            IF JerkFacLocal <= 0.0 THEN
                JerkFacLocal := 0.1;
            END_IF;

            IF TorqueFacLocal <= 0.0 THEN
                TorqueFacLocal := 0.1;
            END_IF;


            //------------------------------------------------
            // Mapping blending
            //------------------------------------------------
            IF (Item.BlendMode = 0)
               OR (Item.BlendRadius <= 0.0)
            THEN

                BufferMode := C_BM_Buffered;
                TransMode  := C_TM_None;

                TransParam[0] := 0.0;
                TransParam[1] := 0.0;

            ELSE

                //------------------------------------------------
                // Dùng giống MoveP đang chạy ổn
                //------------------------------------------------
                BufferMode := GVL.C_BM_BlendingHigh;

                CASE Item.BlendMode OF

                    1:
                        TransMode := C_TM_CornerDistance;

                    2:
                        TransMode := C_TM_StartVelocity;

                ELSE
                    TransMode := C_TM_CornerDistance;

                END_CASE;

                TransParam[0] := Item.BlendRadius;
                TransParam[1] := 0.0;

            END_IF;


            //------------------------------------------------
            // Orientation mode hiện tại của robot
            //------------------------------------------------
			IF AxisGroup.m_id = SCARA_A.m_id THEN
				OrientationMode := POU_MOTION.RBA_OrientationMode;
			ELSE
				OrientationMode := POU_MOTION.RBB_OrientationMode;
			END_IF
            


            //------------------------------------------------
            // Reset outputs cho command mới
            //------------------------------------------------
            Accepted := FALSE;
            Done     := FALSE;
            Error    := FALSE;
            Timeout  := FALSE;
            Aborted  := FALSE;

            ErrorID_Custom := 0;


            State := E_MoveState.MOVE_SEND;

        END_IF;


    //========================================================
    // SEND COMMAND
    //========================================================
    E_MoveState.MOVE_SEND:

        ExecutePulse := TRUE;

        tAcceptTimeout(
            IN := TRUE,
            PT := AcceptTimeoutTime
        );

        State := E_MoveState.MOVE_WAIT_ACCEPT;


    //========================================================
    // WAIT COMMAND ACCEPTED
    //========================================================
    E_MoveState.MOVE_WAIT_ACCEPT:

        //----------------------------------------------------
        // Giữ Execute cho tới khi AxisGroup nhận command
        //----------------------------------------------------
        ExecutePulse := TRUE;

        tAcceptTimeout(
            IN := TRUE,
            PT := AcceptTimeoutTime
        );


        IF fbMoveL.CommandAccepted THEN

            Accepted := TRUE;

            ExecutePulse := FALSE;

            tAcceptTimeout(IN := FALSE);

            tMoveTimeout(
                IN := TRUE,
                PT := MoveTimeoutTime
            );

            State := E_MoveState.MOVE_WAIT_DONE;


        ELSIF fbMoveL.CommandAborted THEN

            ExecutePulse := FALSE;

            Aborted := TRUE;
            Error   := TRUE;

            ErrorID_Custom := 5103;

            tAcceptTimeout(IN := FALSE);

            State := E_MoveState.MOVE_ABORTED;


        ELSIF fbMoveL.Error THEN

            ExecutePulse := FALSE;

            Error   := TRUE;
            ErrorID := fbMoveL.ErrorID;

            ErrorID_Custom := 5104;

            tAcceptTimeout(IN := FALSE);

            State := E_MoveState.MOVE_ERROR;


        ELSIF tAcceptTimeout.Q THEN

            ExecutePulse := FALSE;

            Timeout := TRUE;
            Error   := TRUE;

            ErrorID_Custom := 5105;

            tAcceptTimeout(IN := FALSE);

            State := E_MoveState.MOVE_TIMEOUT;

        END_IF;


    //========================================================
    // WAIT MOTION DONE
    //========================================================
    E_MoveState.MOVE_WAIT_DONE:

        Accepted := TRUE;
        ExecutePulse := FALSE;

        tMoveTimeout(
            IN := TRUE,
            PT := MoveTimeoutTime
        );


        IF fbMoveL.Done THEN

            tMoveTimeout(IN := FALSE);

            //------------------------------------------------
            // Điểm cần check chính xác
            //------------------------------------------------
            IF NOT Item.SkipPositionCheck THEN

                tPosCheckDelay(
                    IN := TRUE,
                    PT := PosCheckDelayTime
                );

                State := E_MoveState.MOVE_CHECK_POS;

            ELSE

                //------------------------------------------------
                // Điểm transition / blending:
                // không bắt Actual Position == Target.
                //------------------------------------------------
                State := E_MoveState.MOVE_DONE;

            END_IF;


        ELSIF fbMoveL.CommandAborted THEN

            Aborted := TRUE;
            Error   := TRUE;

            ErrorID_Custom := 5103;

            tMoveTimeout(IN := FALSE);

            State := E_MoveState.MOVE_ABORTED;


        ELSIF fbMoveL.Error THEN

            Error   := TRUE;
            ErrorID := fbMoveL.ErrorID;

            ErrorID_Custom := 5104;

            tMoveTimeout(IN := FALSE);

            State := E_MoveState.MOVE_ERROR;


        ELSIF tMoveTimeout.Q THEN

            Timeout := TRUE;
            Error   := TRUE;

            ErrorID_Custom := 5106;

            tMoveTimeout(IN := FALSE);

            State := E_MoveState.MOVE_TIMEOUT;

        END_IF;


    //========================================================
    // CHECK FINAL POSITION
    //========================================================
    E_MoveState.MOVE_CHECK_POS:

        Accepted := TRUE;

        tPosCheckDelay(
            IN := TRUE,
            PT := PosCheckDelayTime
        );

        IF tPosCheckDelay.Q THEN

            tPosCheckDelay(IN := FALSE);

            //------------------------------------------------
            // Lưu để debug
            //------------------------------------------------
// 			IF AxisGroup.m_id = SCARA_A.m_id THEN
//             	DonePosition := POU_MONITOR_ROBOT.RB1_POS;
// 			ELSE
// 				DonePosition := POU_MONITOR_ROBOT.RB2_POS;
// 			END_IF;
			IF AxisGroup.m_id = SCARA_A.m_id THEN
            	DonePosition := POU_COORDINATE_.Pos_Out_A_MCS;
			ELSE
				DonePosition := POU_COORDINATE_.Pos_Out_B_MCS;
			END_IF;


            //------------------------------------------------
            // Kiểm tra vị trí cuối MovL
            //------------------------------------------------
            IF F_CheckPositionReached(
                Target := PosBuf,
                //Actual := POU_MONITOR_ROBOT.RB1_POS,
				Actual := DonePosition,
                TolXYZ := GVL.MotionTolXYZ,
                TolR   := GVL.MotionTolR
            )
            THEN

                State := E_MoveState.MOVE_DONE;

            ELSE

                Error := TRUE;

                //------------------------------------------------
                // 5101 = MoveL position not reached
                //------------------------------------------------
                ErrorID_Custom := 5101;

                State := E_MoveState.MOVE_ERROR;

            END_IF;

        END_IF;


    //========================================================
    // DONE
    //========================================================
    E_MoveState.MOVE_DONE:

        Accepted := TRUE;
        Done     := TRUE;

        ExecutePulse := FALSE;

        //----------------------------------------------------
        // Giống FB_RunMoveP đang dùng:
        // giữ Done cho tới khi Manager đã hạ Start
        // và FB gốc đã hoàn toàn rảnh.
        //----------------------------------------------------
        IF NOT Start
           AND NOT fbMoveL.Busy
           AND NOT fbMoveL.Active
        THEN

            State := E_MoveState.MOVE_IDLE;

        END_IF;


    //========================================================
    // ERROR
    //========================================================
    E_MoveState.MOVE_ERROR:

        Error := TRUE;
        ExecutePulse := FALSE;

        IF NOT Start THEN
            State := E_MoveState.MOVE_IDLE;
        END_IF;


    //========================================================
    // TIMEOUT
    //========================================================
    E_MoveState.MOVE_TIMEOUT:

        Error   := TRUE;
        Timeout := TRUE;

        ExecutePulse := FALSE;

        IF NOT Start THEN
            State := E_MoveState.MOVE_IDLE;
        END_IF;


    //========================================================
    // ABORTED
    //========================================================
    E_MoveState.MOVE_ABORTED:

        Error   := TRUE;
        Aborted := TRUE;

        ExecutePulse := FALSE;

        IF NOT Start THEN
            State := E_MoveState.MOVE_IDLE;
        END_IF;

END_CASE;


//============================================================
// GỌI FB GỐC MỖI SCAN
//============================================================
fbMoveL(
    AxisGroup := AxisGroup,

    Execute := ExecutePulse,

    Position := PosBuf,

    Velocity     := Vel,
    Acceleration := Acc,
    Deceleration := Dec,
    Jerk         := Jerk,

    CoordSystem := CoordSystem,

    BufferMode          := BufferMode,
    TransitionMode      := TransMode,
    TransitionParameter := TransParam,

    OrientationMode := OrientationMode,

    VelFactor    := VelFacLocal,
    AccFactor    := AccFacLocal,
    JerkFactor   := JerkFacLocal,
    TorqueFactor := TorqueFacLocal
);


//============================================================
// PHẢN HỒI TRẠNG THÁI FB GỐC
//============================================================
Busy   := fbMoveL.Busy;
Active := fbMoveL.Active;

END_FUNCTION_BLOCK

// Just_Motion_Control_x86_64_Linux_SM_WV/Application/FB_/FB_RunMoveC
FUNCTION_BLOCK FB_RunMoveC
VAR_INPUT
    Start : BOOL;
    Item  : ST_MotionQueueItem;

    //--------------------------------------------------------
    // Điểm trung gian nằm trên cung
    //--------------------------------------------------------
    MidPosition : SMC_POS_REF;

    //--------------------------------------------------------
    // Điểm cuối cung
    //--------------------------------------------------------
    EndPosition : SMC_POS_REF;

    CoordSystem : SMC_COORD_SYSTEM;

    AcceptTimeoutTime : TIME := T#2S;
    MoveTimeoutTime   : TIME := T#100S;
    PosCheckDelayTime : TIME := T#13MS;
END_VAR

VAR_IN_OUT
    AxisGroup : AXIS_GROUP_REF_SM3;
    //Release   : BOOL;
END_VAR

VAR_OUTPUT
    Accepted       : BOOL;
    Done           : BOOL;
    Busy           : BOOL;
    Active         : BOOL;
    Error          : BOOL;
    Timeout        : BOOL;
    Aborted        : BOOL;

    ErrorID        : SMC_ERROR;
    ErrorID_Custom : INT;

    State          : E_MoveState;
END_VAR

VAR
    //--------------------------------------------------------
    // SoftMotion FB
    //--------------------------------------------------------
    fbMoveC : MC_MoveCircularAbsolute;

    //--------------------------------------------------------
    // Timer
    //--------------------------------------------------------
    tAcceptTimeout : TON;
    tMoveTimeout   : TON;
    tPosCheckDelay : TON;

    //--------------------------------------------------------
    // Execute
    //--------------------------------------------------------
    StartEdge    : BOOL;
    LastStart    : BOOL;
    ExecutePulse : BOOL;

    //--------------------------------------------------------
    // Position buffer
    //--------------------------------------------------------
    MidBuf       : SMC_POS_REF;
    EndBuf       : SMC_POS_REF;
    DonePosition : SMC_POS_REF;

    //--------------------------------------------------------
    // Path dynamics
    //--------------------------------------------------------
    Vel  : LREAL;
    Acc  : LREAL;
    Dec  : LREAL;
    Jerk : LREAL;

    //--------------------------------------------------------
    // Circular parameters
    //--------------------------------------------------------
    CircModeLocal :
        SM3_Robotics.SMC_CIRC_MODE;

    PathChoiceLocal :
        SM3_Robotics.MC_CIRC_PATHCHOICE;

    //--------------------------------------------------------
    // Blending
    //--------------------------------------------------------
    BufferMode :
        SM3_Robotics.MC_BUFFER_MODE;

    TransMode :
        SM3_Robotics.MC_TRANSITION_MODE;

    TransParam :
        ARRAY[0..(SMC_RCNST.MAX_TRANS_PARAMS - 1)] OF LREAL
        := [0.0, 0.0];

    //--------------------------------------------------------
    // Orientation
    //--------------------------------------------------------
    OrientationMode :
        SM3_Robotics.SMC_ORIENTATION_MODE;

    //--------------------------------------------------------
    // Factor
    //--------------------------------------------------------
    VelFacLocal    : LREAL;
    AccFacLocal    : LREAL;
    JerkFacLocal   : LREAL;
    TorqueFacLocal : LREAL;
END_VAR

VAR CONSTANT
    C_BM_Buffered :
        SM3_Robotics.MC_BUFFER_MODE := 1;

    C_TM_CornerDistance :
        SM3_Robotics.MC_TRANSITION_MODE := 2;

    C_TM_None :
        SM3_Robotics.MC_TRANSITION_MODE := 0;

    C_TM_StartVelocity :
        SM3_Robotics.MC_TRANSITION_MODE := 1;
END_VAR

//============================================================
// FB_RunMoveC
//
// Quỹ đạo:
// Current Position → MidPosition → EndPosition
//
// CircMode = BORDER:
// MidPosition là điểm nằm trên cung.
//
// Cơ chế Accepted / Done / Error giống FB_RunMoveP.
//============================================================


//------------------------------------------------------------
// Start edge
//------------------------------------------------------------
StartEdge := Start AND NOT LastStart;
LastStart := Start;


//------------------------------------------------------------
// Execute mặc định FALSE
//------------------------------------------------------------
ExecutePulse := FALSE;


//============================================================
// STATE MACHINE
//============================================================
CASE State OF


    //========================================================
    // IDLE
    //========================================================
    E_MoveState.MOVE_IDLE:

        Accepted := FALSE;
        Done     := FALSE;
        Error    := FALSE;
        Timeout  := FALSE;
        Aborted  := FALSE;

        //Release := FALSE;

        ErrorID_Custom := 0;

        //----------------------------------------------------
        // Reset timer
        //----------------------------------------------------
        tAcceptTimeout(IN := FALSE);
        tMoveTimeout(IN := FALSE);
        tPosCheckDelay(IN := FALSE);


        //----------------------------------------------------
        // Chỉ nhận command khi FB rảnh
        //----------------------------------------------------
        IF Start
           AND NOT fbMoveC.Busy
           AND NOT fbMoveC.Active
        THEN

            //------------------------------------------------
            // Chốt điểm giữa và điểm cuối
            //------------------------------------------------
            MidBuf := MidPosition;
            EndBuf := EndPosition;


            //------------------------------------------------
            // Dynamics
            //------------------------------------------------
           	
			IF Item.Speed > 0.0 THEN
                Vel := Item.Speed;
            ELSE
				IF AxisGroup.m_id = SCARA_A.m_id THEN
                	Vel := GVL.A_CurrentMotionParam.Speed;
				ELSE
					Vel := GVL.B_CurrentMotionParam.Speed;
				END_IF
            END_IF;

            IF AxisGroup.m_id = SCARA_A.m_id THEN
				IF Item.Acceleration > 0.0 THEN Acc := Item.Acceleration; ELSE Acc := GVL_1.DATA_RB_A.MOTION_ACC; END_IF;
				IF Item.Deceleration > 0.0 THEN Dec := Item.Deceleration; ELSE Dec := GVL_1.DATA_RB_A.MOTION_DEC; END_IF;
				IF Item.Jerk > 0.0 THEN Jerk := Item.Jerk; ELSE Jerk := GVL_1.DATA_RB_A.MOTION_JERK; END_IF;
			ELSE
				IF Item.Acceleration > 0.0 THEN Acc := Item.Acceleration; ELSE Acc := GVL_1.DATA_RB_B.MOTION_ACC; END_IF;
				IF Item.Deceleration > 0.0 THEN Dec := Item.Deceleration; ELSE Dec := GVL_1.DATA_RB_B.MOTION_DEC; END_IF;
				IF Item.Jerk > 0.0 THEN Jerk := Item.Jerk; ELSE Jerk := GVL_1.DATA_RB_B.MOTION_JERK; END_IF;
			END_IF


            //------------------------------------------------
            // Fallback
            //------------------------------------------------
            IF Vel <= 0.0 THEN
                Vel := 100.0;
            END_IF;

            IF Acc <= 0.0 THEN
                Acc := 1000.0;
            END_IF;

            IF Dec <= 0.0 THEN
                Dec := 1000.0;
            END_IF;

            IF Jerk <= 0.0 THEN
                Jerk := 10000.0;
            END_IF;


            //------------------------------------------------
            // Factor
            //------------------------------------------------
            IF AxisGroup.m_id = SCARA_A.m_id THEN
				VelFacLocal    := GVL_1.DATA_RB_A.Fac_Vel;
				AccFacLocal    := GVL_1.DATA_RB_A.Fac_Acc;
				JerkFacLocal   := GVL_1.DATA_RB_A.Fac_Jerk;
				TorqueFacLocal := GVL_1.DATA_RB_A.Fac_Torque;
			ELSE
				VelFacLocal    := GVL_1.DATA_RB_B.Fac_Vel;
				AccFacLocal    := GVL_1.DATA_RB_B.Fac_Acc;
				JerkFacLocal   := GVL_1.DATA_RB_B.Fac_Jerk;
				TorqueFacLocal := GVL_1.DATA_RB_B.Fac_Torque;
			END_IF

            IF VelFacLocal <= 0.0 THEN
                VelFacLocal := 0.1;
            END_IF;

            IF AccFacLocal <= 0.0 THEN
                AccFacLocal := 0.1;
            END_IF;

            IF JerkFacLocal <= 0.0 THEN
                JerkFacLocal := 0.1;
            END_IF;

            IF TorqueFacLocal <= 0.0 THEN
                TorqueFacLocal := 0.1;
            END_IF;


            //------------------------------------------------
            // CIRCULAR MODE
            //
            // MidPosition được dạy như điểm nằm trên cung.
            //------------------------------------------------
            CircModeLocal :=
                SM3_Robotics.SMC_CIRC_MODE.BORDER;

            //------------------------------------------------
            // BORDER không dùng PathChoice,
            // nhưng input FB vẫn phải có giá trị hợp lệ.
            //------------------------------------------------
            PathChoiceLocal :=
                SM3_Robotics.MC_CIRC_PATHCHOICE.CLOCKWISE;


            //------------------------------------------------
            // Mapping Blend giống MoveP / MoveL
            //------------------------------------------------
            IF (Item.BlendMode = 0)
               OR (Item.BlendRadius <= 0.0)
            THEN

                BufferMode := C_BM_Buffered;
                TransMode  := C_TM_None;

                TransParam[0] := 0.0;
                TransParam[1] := 0.0;

            ELSE

                BufferMode := GVL.C_BM_BlendingHigh;

                CASE Item.BlendMode OF

                    1:
                        TransMode := C_TM_CornerDistance;

                    2:
                        TransMode := C_TM_StartVelocity;

                ELSE
                    TransMode := C_TM_CornerDistance;

                END_CASE;

                TransParam[0] := Item.BlendRadius;
                TransParam[1] := 0.0;

            END_IF;


            //------------------------------------------------
            // Orientation
            //------------------------------------------------
            IF AxisGroup.m_id = SCARA_A.m_id THEN
				OrientationMode := POU_MOTION.RBA_OrientationMode;
			ELSE
				OrientationMode := POU_MOTION.RBB_OrientationMode;
			END_IF


            //------------------------------------------------
            // Reset outputs
            //------------------------------------------------
            Accepted := FALSE;
            Done     := FALSE;
            Error    := FALSE;
            Timeout  := FALSE;
            Aborted  := FALSE;

            ErrorID_Custom := 0;


            State := E_MoveState.MOVE_SEND;

        END_IF;


    //========================================================
    // SEND COMMAND
    //========================================================
    E_MoveState.MOVE_SEND:

        ExecutePulse := TRUE;

        tAcceptTimeout(
            IN := TRUE,
            PT := AcceptTimeoutTime
        );

        State := E_MoveState.MOVE_WAIT_ACCEPT;


    //========================================================
    // WAIT ACCEPT
    //========================================================
    E_MoveState.MOVE_WAIT_ACCEPT:

        ExecutePulse := TRUE;

        tAcceptTimeout(
            IN := TRUE,
            PT := AcceptTimeoutTime
        );


        IF fbMoveC.CommandAccepted THEN

            Accepted := TRUE;

            ExecutePulse := FALSE;

            tAcceptTimeout(IN := FALSE);

            tMoveTimeout(
                IN := TRUE,
                PT := MoveTimeoutTime
            );

            State := E_MoveState.MOVE_WAIT_DONE;


        ELSIF fbMoveC.CommandAborted THEN

            ExecutePulse := FALSE;

            Aborted := TRUE;
            Error   := TRUE;

            ErrorID_Custom := 5203;

            tAcceptTimeout(IN := FALSE);

            State := E_MoveState.MOVE_ABORTED;


        ELSIF fbMoveC.Error THEN

            ExecutePulse := FALSE;

            Error   := TRUE;
            ErrorID := fbMoveC.ErrorID;

            ErrorID_Custom := 5204;

            tAcceptTimeout(IN := FALSE);

            State := E_MoveState.MOVE_ERROR;


        ELSIF tAcceptTimeout.Q THEN

            ExecutePulse := FALSE;

            Timeout := TRUE;
            Error   := TRUE;

            ErrorID_Custom := 5205;

            tAcceptTimeout(IN := FALSE);

            State := E_MoveState.MOVE_TIMEOUT;

        END_IF;


    //========================================================
    // WAIT DONE
    //========================================================
    E_MoveState.MOVE_WAIT_DONE:

        Accepted := TRUE;
        ExecutePulse := FALSE;

        tMoveTimeout(
            IN := TRUE,
            PT := MoveTimeoutTime
        );


        IF fbMoveC.Done THEN

            tMoveTimeout(IN := FALSE);

            //------------------------------------------------
            // MovC chỉ check vị trí cuối EndBuf.
            //
            // MidBuf tuyệt đối không check vì đó chỉ là điểm
            // dùng để xác định hình học của cung.
            //------------------------------------------------
            IF NOT Item.SkipPositionCheck THEN

                tPosCheckDelay(
                    IN := TRUE,
                    PT := PosCheckDelayTime
                );

                State := E_MoveState.MOVE_CHECK_POS;

            ELSE

                State := E_MoveState.MOVE_DONE;

            END_IF;


        ELSIF fbMoveC.CommandAborted THEN

            Aborted := TRUE;
            Error   := TRUE;

            ErrorID_Custom := 5203;

            tMoveTimeout(IN := FALSE);

            State := E_MoveState.MOVE_ABORTED;


        ELSIF fbMoveC.Error THEN

            Error   := TRUE;
            ErrorID := fbMoveC.ErrorID;

            ErrorID_Custom := 5204;

            tMoveTimeout(IN := FALSE);

            State := E_MoveState.MOVE_ERROR;


        ELSIF tMoveTimeout.Q THEN

            Timeout := TRUE;
            Error   := TRUE;

            ErrorID_Custom := 5206;

            tMoveTimeout(IN := FALSE);

            State := E_MoveState.MOVE_TIMEOUT;

        END_IF;


    //========================================================
    // CHECK END POSITION
    //========================================================
    E_MoveState.MOVE_CHECK_POS:

        Accepted := TRUE;

        tPosCheckDelay(
            IN := TRUE,
            PT := PosCheckDelayTime
        );

        IF tPosCheckDelay.Q THEN

            tPosCheckDelay(IN := FALSE);

            //------------------------------------------------
            // Lưu để debug
            //------------------------------------------------
//             IF AxisGroup.m_id = SCARA_A.m_id THEN
//             	DonePosition := POU_MONITOR_ROBOT.RB1_POS;
// 			ELSE
// 				DonePosition := POU_MONITOR_ROBOT.RB2_POS;
// 			END_IF;
			
			IF AxisGroup.m_id = SCARA_A.m_id THEN
            	DonePosition := POU_COORDINATE_.Pos_Out_A_MCS;
			ELSE
				DonePosition := POU_COORDINATE_.Pos_Out_B_MCS;
			END_IF;



            //------------------------------------------------
            // Với MoveC chỉ kiểm tra END POINT.
            //------------------------------------------------
            IF F_CheckPositionReached(
                Target := EndBuf,
                //Actual := POU_MONITOR_ROBOT.RB1_POS,
				Actual := DonePosition,
                TolXYZ := GVL.MotionTolXYZ,
                TolR   := GVL.MotionTolR
            )
            THEN

                State := E_MoveState.MOVE_DONE;

            ELSE

                Error := TRUE;

                //------------------------------------------------
                // 5201 = Circular end position not reached
                //------------------------------------------------
                ErrorID_Custom := 5201;

                State := E_MoveState.MOVE_ERROR;

            END_IF;

        END_IF;


    //========================================================
    // DONE
    //========================================================
    E_MoveState.MOVE_DONE:

        Accepted := TRUE;
        Done     := TRUE;

        ExecutePulse := FALSE;

        IF NOT Start
           AND NOT fbMoveC.Busy
           AND NOT fbMoveC.Active
        THEN

            State := E_MoveState.MOVE_IDLE;

        END_IF;


    //========================================================
    // ERROR
    //========================================================
    E_MoveState.MOVE_ERROR:

        Error := TRUE;
        ExecutePulse := FALSE;

        IF NOT Start THEN
            State := E_MoveState.MOVE_IDLE;
        END_IF;


    //========================================================
    // TIMEOUT
    //========================================================
    E_MoveState.MOVE_TIMEOUT:

        Error   := TRUE;
        Timeout := TRUE;

        ExecutePulse := FALSE;

        IF NOT Start THEN
            State := E_MoveState.MOVE_IDLE;
        END_IF;


    //========================================================
    // ABORTED
    //========================================================
    E_MoveState.MOVE_ABORTED:

        Error   := TRUE;
        Aborted := TRUE;

        ExecutePulse := FALSE;

        IF NOT Start THEN
            State := E_MoveState.MOVE_IDLE;
        END_IF;

END_CASE;


//============================================================
// GỌI FB GỐC MỖI SCAN
//============================================================
fbMoveC(
    AxisGroup := AxisGroup,

    Execute := ExecutePulse,

    //--------------------------------------------------------
    // Dùng BORDER:
    // MidBuf là điểm nằm trên cung.
    //--------------------------------------------------------
    CircMode := CircModeLocal,
    AuxPoint := MidBuf,
    EndPoint := EndBuf,

    PathChoice := PathChoiceLocal,

    Velocity     := Vel,
    Acceleration := Acc,
    Deceleration := Dec,
    Jerk         := Jerk,

    CoordSystem := CoordSystem,

    BufferMode          := BufferMode,
    TransitionMode      := TransMode,
    TransitionParameter := TransParam,

    OrientationMode := OrientationMode,

    VelFactor    := VelFacLocal,
    AccFactor    := AccFacLocal,
    JerkFactor   := JerkFacLocal,
    TorqueFactor := TorqueFacLocal
);


//============================================================
// PHẢN HỒI FB GỐC
//============================================================
Busy   := fbMoveC.Busy;
Active := fbMoveC.Active;

END_FUNCTION_BLOCK

// Just_Motion_Control_x86_64_Linux_SM_WV/Application/FB_/Vision/FB_VisionAlign
FUNCTION_BLOCK FB_VisionAlign
VAR_INPUT
    Enable : BOOL;                              // Cho phép FB hoạt động.
    Start : BOOL;                               // Bắt đầu một lần Align.
    CameraID : UINT;                            // Camera sử dụng.
    JobID : UINT;                               // Job Vision Align.
END_VAR

VAR_OUTPUT
    Busy : BOOL;                                // Đang chạy.
    Done : BOOL;                                // Hoàn thành.
    Error : BOOL;                               // Có lỗi.
    ErrorID : INT;                              // Mã lỗi.
    State : INT;                                // State monitor.

    HeaderOK : BOOL;                            // Đã nhận Header hợp lệ.
    TriggerID : UDINT;                          // TriggerID của Result.

    VisionX : REAL;                             // X Vision trả về.
    VisionY : REAL;                             // Y Vision trả về.
    VisionZ : REAL;                             // Z Vision trả về.
    VisionA : REAL;                             // Theta Vision trả về.
    VisionScore : REAL;                         // Score Vision.
    VisionFeatureID : UINT;                     // FeatureID Vision.

    ResultValid : BOOL;                         // Valid từ Vision.
    ResultStatus : E_VisionResultStatus;        // Status Vision.
END_VAR

VAR
    StartOld : BOOL;                            // Start scan trước.
    xStartVision : BOOL;                        // Start FB VisionGetResult.

    fbVisionGetResult : FB_VisionGetResult;     // FB Trigger + nhận Result.
END_VAR

//=============================================================================
// FB_VisionAlign - SIMPLE VERSION
//-----------------------------------------------------------------------------
// FB này không tự xử lý Modbus.
// Không tự gọi FB_TriggerVS / FB_VisionWaitResult.
// Toàn bộ Trigger + nhận Result giao cho FB_VisionGetResult.
//=============================================================================


//=============================================================================
// CALL FB VISION GET RESULT
//=============================================================================
fbVisionGetResult(
    Enable := Enable,
    Start := xStartVision,
    CameraID := CameraID,
    JobID := JobID,
    Application := E_VisionApplication.VIS_APP_ALIGN
);


//=============================================================================
// RESET
//=============================================================================
IF NOT Enable THEN
    State := 0;
    StartOld := FALSE;
    xStartVision := FALSE;

    Busy := FALSE;
    Done := FALSE;
    Error := FALSE;
    ErrorID := 0;

    HeaderOK := FALSE;
    TriggerID := 0;

    VisionX := 0.0;
    VisionY := 0.0;
    VisionZ := 0.0;
    VisionA := 0.0;
    VisionScore := 0.0;
    VisionFeatureID := 0;

    ResultValid := FALSE;
    ResultStatus := E_VisionResultStatus.VIS_RESULT_NONE;

    RETURN;
END_IF;


//=============================================================================
// STATE MACHINE
//=============================================================================
CASE State OF

    //=========================================================================
    // 0 - IDLE
    //=========================================================================
    0:
        Busy := FALSE;
        Done := FALSE;
        Error := FALSE;
        ErrorID := 0;

        xStartVision := FALSE;
        HeaderOK := FALSE;

        IF Start AND NOT StartOld THEN
            Busy := TRUE;

            xStartVision := TRUE;

            State := 10;
        END_IF;


    //=========================================================================
    // 10 - WAIT VISION RESULT
    //=========================================================================
    10:
        Busy := TRUE;

        IF fbVisionGetResult.Error THEN
            xStartVision := FALSE;

            Error := TRUE;
            ErrorID := fbVisionGetResult.ErrorID;

            State := 900;

        ELSIF fbVisionGetResult.Done THEN
            xStartVision := FALSE;

            State := 20;
        END_IF;


    //=========================================================================
    // 20 - COPY VISION RESULT
    //=========================================================================
    20:
        HeaderOK := fbVisionGetResult.HeaderOK;
        TriggerID := fbVisionGetResult.TriggerID;

        VisionX := fbVisionGetResult.X;
        VisionY := fbVisionGetResult.Y;
        VisionZ := fbVisionGetResult.Z;
        VisionA := fbVisionGetResult.A;
        VisionScore := fbVisionGetResult.Score;
        VisionFeatureID := fbVisionGetResult.FeatureID;

        ResultValid := fbVisionGetResult.ResultValid;
        ResultStatus := fbVisionGetResult.ResultStatus;

        State := 30;


    //=========================================================================
    // 30 - ALIGN RESULT READY
    //-------------------------------------------------------------------------
    // Hiện tại chưa xử lý Transform / Correction.
    // Chỉ xác nhận đã nhận được dữ liệu Vision.
    //=========================================================================
    30:
        IF HeaderOK THEN
            Busy := FALSE;
            Done := TRUE;

            State := 100;
        ELSE
            Error := TRUE;
            ErrorID := 301;                  // Không có Header hợp lệ.

            State := 900;
        END_IF;


    //=========================================================================
    // 100 - DONE
    //=========================================================================
    100:
        Busy := FALSE;
        Done := TRUE;

        IF NOT Start THEN
            State := 0;
        END_IF;


    //=========================================================================
    // 900 - ERROR
    //=========================================================================
    900:
        Busy := FALSE;
        Done := FALSE;

        xStartVision := FALSE;

        IF NOT Start THEN
            Error := FALSE;
            ErrorID := 0;

            State := 0;
        END_IF;

END_CASE;


//=============================================================================
// SAVE START
//=============================================================================
StartOld := Start;

END_FUNCTION_BLOCK

// Just_Motion_Control_x86_64_Linux_SM_WV/Application/FB_/Vision/FB_VisionGetResult
FUNCTION_BLOCK FB_VisionGetResult
VAR_INPUT
    Enable : BOOL;                              // Cho phép FB hoạt động.
    Start : BOOL;                               // Cạnh lên bắt đầu một lần đọc Vision.
    CameraID : UINT;                            // Camera sử dụng.
    JobID : UINT;                               // JobID Vision.
    Application : E_VisionApplication;          // Application Vision.
END_VAR

VAR_OUTPUT
    Busy : BOOL;                                // Đang thực hiện.
    Done : BOOL;                                // Đã nhận Result thành công.
    Error : BOOL;                               // Có lỗi.
    ErrorID : INT;                              // Mã lỗi.

    State : INT;                                // State để monitor.

    TriggerID : UDINT;                          // TriggerID của lần chụp.

    HeaderOK : BOOL;                            // TRUE khi Header Result hợp lệ.

    ResultValid : BOOL;                         // Bit Valid của dữ liệu Vision.
    ResultStatus : E_VisionResultStatus;        // ResultStatus Vision.
    ResultCode : UINT;                          // ResultCode Vision.
    VisionErrorCode : UINT;                     // ErrorCode Vision.

    X : REAL;                                   // X Vision trả về.
    Y : REAL;                                   // Y Vision trả về.
    Z : REAL;                                   // Z Vision trả về.
    A : REAL;                                   // Theta / Angle Vision trả về.
    Score : REAL;                               // Score Vision.
    FeatureID : UINT;                           // FeatureID Vision.
END_VAR

VAR
    StartOld : BOOL;                            // Start scan trước.

    xStartTrigger : BOOL;                       // Start nội bộ cho Trigger.
    xStartWaitResult : BOOL;                    // Start nội bộ cho WaitResult.

    fbTriggerVS : FB_TriggerVS;                 // FB Trigger đã test.
    fbWaitResult : FB_VisionWaitResult;         // FB WaitResult đã test.
END_VAR

//=============================================================================
// FB_VisionGetResult
//-----------------------------------------------------------------------------
// Chức năng đơn giản:
// 1. Trigger Vision.
// 2. Chờ Vision trả Result.
// 3. Khi Header hợp lệ và đúng TriggerID thì copy dữ liệu ra Output.
// 4. Không kiểm tra Offset / Tolerance / Motion.
//=============================================================================


//=============================================================================
// CALL TRIGGER
//=============================================================================
fbTriggerVS(
    Enable := Enable,
    Start := xStartTrigger,
    CameraID := CameraID,
    JobID := JobID,
    Application := Application,
    count_Vs_Align_max := GVL.g_aVisionConfig[CameraID].MaxRetry,
    T_Delay_Trigger_time := TO_INT(GVL.g_aVisionConfig[CameraID].TriggerTimeout),
    Trigger_Again := FALSE,
    Pass_Triger_VS_NG := FALSE,
    Mode_ByPass_VS := FALSE
);

TriggerID := fbTriggerVS.CurrentTriggerID;


//=============================================================================
// CALL WAIT RESULT
//=============================================================================
fbWaitResult(
    Enable := Enable,
    Start := xStartWaitResult,
    CameraID := CameraID,
    ExpectedTriggerID := TriggerID,
    ExpectedJobID := JobID,
    ExpectedApplication := Application
);


//=============================================================================
// DISABLE / RESET
//=============================================================================
IF NOT Enable THEN
    State := 0;
    StartOld := FALSE;

    Busy := FALSE;
    Done := FALSE;
    Error := FALSE;
    ErrorID := 0;

    xStartTrigger := FALSE;
    xStartWaitResult := FALSE;

    HeaderOK := FALSE;

    ResultValid := FALSE;
    ResultStatus := E_VisionResultStatus.VIS_RESULT_NONE;
    ResultCode := 0;
    VisionErrorCode := 0;

    X := 0.0;
    Y := 0.0;
    Z := 0.0;
    A := 0.0;
    Score := 0.0;
    FeatureID := 0;

    RETURN;
END_IF;


//=============================================================================
// STATE MACHINE
//=============================================================================
CASE State OF

    //=========================================================================
    // 0 - IDLE
    //=========================================================================
    0:
        Busy := FALSE;
        Done := FALSE;
        Error := FALSE;
        ErrorID := 0;

        xStartTrigger := FALSE;
        xStartWaitResult := FALSE;

        HeaderOK := FALSE;

        IF Start AND NOT StartOld THEN
            Busy := TRUE;
            xStartTrigger := TRUE;
            State := 10;
        END_IF;


    //=========================================================================
    // 10 - WAIT TRIGGER DONE
    //=========================================================================
    10:
        Busy := TRUE;

        IF fbTriggerVS.Error THEN
            xStartTrigger := FALSE;

            Error := TRUE;
            ErrorID := 100 + fbTriggerVS.ErrorID;
            State := 900;

        ELSIF fbTriggerVS.DoneAll THEN
            xStartTrigger := FALSE;

            xStartWaitResult := TRUE;
            State := 20;
        END_IF;


    //=========================================================================
    // 20 - WAIT RESULT
    //=========================================================================
    20:
        Busy := TRUE;

        IF fbWaitResult.Error THEN
            xStartWaitResult := FALSE;

            Error := TRUE;
            ErrorID := 200 + fbWaitResult.ErrorID;
            State := 900;

        ELSIF fbWaitResult.Done THEN
            xStartWaitResult := FALSE;

            State := 30;
        END_IF;


    //=========================================================================
    // 30 - COPY RESULT
    //=========================================================================
    30:
        // Header đã được FB_WaitResult xác nhận đúng TriggerID / JobID / App.
        HeaderOK := TRUE;

        ResultValid := fbWaitResult.ResultValid;
        ResultStatus := fbWaitResult.ResultStatus;
        ResultCode := fbWaitResult.ResultCode;
        VisionErrorCode := fbWaitResult.VisionErrorCode;

        X := fbWaitResult.ResultX;
        Y := fbWaitResult.ResultY;
        Z := fbWaitResult.ResultZ;
        A := fbWaitResult.ResultA;
        Score := fbWaitResult.ResultScore;
        FeatureID := fbWaitResult.ResultFeatureID;

        Busy := FALSE;
        Done := TRUE;

        State := 100;


    //=========================================================================
    // 100 - DONE
    //=========================================================================
    100:
        Busy := FALSE;
        Done := TRUE;

        IF NOT Start THEN
            State := 0;
        END_IF;


    //=========================================================================
    // 900 - ERROR
    //=========================================================================
    900:
        Busy := FALSE;
        Done := FALSE;

        xStartTrigger := FALSE;
        xStartWaitResult := FALSE;

        IF NOT Start THEN
            Error := FALSE;
            ErrorID := 0;
            State := 0;
        END_IF;

END_CASE;

StartOld := Start;

END_FUNCTION_BLOCK

// Just_Motion_Control_x86_64_Linux_SM_WV/Application/FB_/FB_MotionQueuePush_B
FUNCTION_BLOCK FB_MotionQueuePush_B
VAR_INPUT
	Item : ST_MotionQueueItem;
    Execute : BOOL;
END_VAR
VAR_OUTPUT
	Done : BOOL;
    Error : BOOL;
	Busy  : BOOL;
END_VAR
VAR
	ExecuteOld  : BOOL;
	ExecuteRise : BOOL;
END_VAR

//====================================================
// FB_MotionQueuePush
// Execute = TRUE  -> Push đúng 1 lần
// Done/Error giữ đến khi Execute = FALSE
//====================================================

IF NOT Execute THEN

    Done := FALSE;
    Error := FALSE;
    Busy := FALSE;

ELSE

    IF NOT Busy THEN

        Busy := TRUE;

        IF GVL.B_MotionCount >= 20 THEN

            Error := TRUE;
            Done := FALSE;

        ELSE

            GVL.B_MotionQueue[GVL.B_MotionTail] := Item;

            GVL.B_MotionTail := GVL.B_MotionTail + 1;

            IF GVL.B_MotionTail > 20 THEN
                GVL.B_MotionTail := 1;
            END_IF;

            GVL.B_MotionCount := GVL.B_MotionCount + 1;

            Done := TRUE;
            Error := FALSE;

        END_IF;

    END_IF;

END_IF;

END_FUNCTION_BLOCK

// Just_Motion_Control_x86_64_Linux_SM_WV/Application/FB_/FB_MotionQueuePop_B
FUNCTION_BLOCK FB_MotionQueuePop_B
VAR_INPUT
	Execute : BOOL;
END_VAR
VAR_OUTPUT
	Item  : ST_MotionQueueItem;
    Done  : BOOL;
    Empty : BOOL;
	Busy  : BOOL;
END_VAR
VAR
	ExecuteOld  : BOOL;
	ExecuteRise : BOOL;
END_VAR

IF NOT Execute THEN

    Done := FALSE;
    Empty := FALSE;
    Busy := FALSE;

ELSE

    IF NOT Busy THEN

        Busy := TRUE;

        IF GVL.B_MotionCount <= 0 THEN

            Empty := TRUE;
            Done := FALSE;

        ELSE

            Item := GVL.B_MotionQueue[GVL.B_MotionHead];

            GVL.B_MotionHead := GVL.B_MotionHead + 1; // Tang gia tri len 1 sau khi lay

            IF GVL.B_MotionHead > 20 THEN // Nếu Head vượt quá 20 thì quay lại 1
                GVL.B_MotionHead := 1;
            END_IF;

            GVL.B_MotionCount := GVL.B_MotionCount - 1; // giam so luong phan di trong queue di 1

            Done := TRUE;
            Empty := FALSE;

        END_IF;

    END_IF;

END_IF;

END_FUNCTION_BLOCK

// Just_Motion_Control_x86_64_Linux_SM_WV/Application/FC_/F_IsMotionCmd
FUNCTION F_IsMotionCmd : BOOL // Kiem tra xem phai la motion cmd khong
VAR_INPUT
	Cmd : E_RobotCmd;
END_VAR
VAR
END_VAR

CASE Cmd OF
    E_RobotCmd.CMD_MovP,
    E_RobotCmd.CMD_MovL,
    E_RobotCmd.CMD_MovC:
        F_IsMotionCmd := TRUE;
ELSE
    F_IsMotionCmd := FALSE;
END_CASE

END_FUNCTION

// Just_Motion_Control_x86_64_Linux_SM_WV/Application/FC_/RBA/F_EvalCondition_A
FUNCTION F_EvalCondition_A : BOOL
VAR_INPUT
    CondNo : INT;
END_VAR

VAR
    i : INT;
    rowResult : BOOL;
    finalResult : BOOL;
    firstRow : BOOL;
END_VAR

IF (CondNo < 1) OR (CondNo > 100) THEN
    F_EvalCondition_A := FALSE;
    RETURN;
END_IF;

IF NOT GVL_1.Condition_Cr_A[CondNo].Enable THEN
    F_EvalCondition_A := FALSE;
    RETURN;
END_IF;

firstRow := TRUE;
finalResult := FALSE;

FOR i := 1 TO 10 DO

    IF GVL_1.Condition_Cr_A[CondNo].Row[i].Enable THEN

        rowResult := F_EvalCondRow_A(GVL_1.Condition_Cr_A[CondNo].Row[i]);

        IF firstRow THEN
            finalResult := rowResult;
            firstRow := FALSE;
        ELSE
            CASE GVL_1.Condition_Cr_A[CondNo].Row[i - 1].LinkNext OF
                1: finalResult := finalResult AND rowResult;
                2: finalResult := finalResult OR rowResult;
            ELSE
                finalResult := finalResult AND rowResult;
            END_CASE;
        END_IF;

    END_IF;

END_FOR;

GVL_1.Condition_Cr_A[CondNo].Result := finalResult;
F_EvalCondition_A := finalResult;

END_FUNCTION

// Just_Motion_Control_x86_64_Linux_SM_WV/Application/FC_/RBA/F_EvalCondRow_A
FUNCTION F_EvalCondRow_A : BOOL
VAR_INPUT
    Row : ST_ConditionRow;
END_VAR

VAR
    actualValue : LREAL;
END_VAR

IF NOT Row.Enable THEN
    F_EvalCondRow_A := TRUE;
    RETURN;
END_IF;

actualValue := F_GetCondValue_A(
    Source := Row.Source,
    Index  := Row.Index
);

CASE Row.Operator OF
    1: F_EvalCondRow_A := actualValue = Row.SetValue;
    2: F_EvalCondRow_A := actualValue <> Row.SetValue;
    3: F_EvalCondRow_A := actualValue > Row.SetValue;
    4: F_EvalCondRow_A := actualValue >= Row.SetValue;
    5: F_EvalCondRow_A := actualValue < Row.SetValue;
    6: F_EvalCondRow_A := actualValue <= Row.SetValue;
ELSE
    F_EvalCondRow_A := FALSE;
END_CASE;

END_FUNCTION

// Just_Motion_Control_x86_64_Linux_SM_WV/Application/FC_/RBA/F_GetCondValue_A
FUNCTION F_GetCondValue_A : DINT
VAR_INPUT
    Source : INT;
    Index  : INT;
END_VAR

CASE Source OF
	0:
    1: // DI
        IF GVL.X[Index] THEN
            F_GetCondValue_A := 1;
        ELSE
            F_GetCondValue_A := 0;
        END_IF;

    2: // DO
        IF GVL.Y[Index] THEN
            F_GetCondValue_A := 1;
        ELSE
            F_GetCondValue_A := 0;
        END_IF;

//     3: // REG
//         F_GetCondValue_A := GVL.A_Reg[Index];
// 
//     4: // VAR
//         F_GetCondValue_A := GVL.A_Var[Index];

ELSE
    F_GetCondValue_A := 0;

END_CASE;

END_FUNCTION

// Just_Motion_Control_x86_64_Linux_SM_WV/Application/FC_/RBA/F_FindElseOrEndIf_A
FUNCTION F_FindElseOrEndIf_A : INT
VAR_INPUT
    StartStep : INT;
END_VAR

VAR
    i : INT;
    depth : INT;
    cmd : E_RobotCmd;
END_VAR

//====================================================
// Tìm ELSE hoặc END_IF tương ứng với IF tại StartStep
// Có hỗ trợ IF lồng nhau
//====================================================

depth := 0;

FOR i := StartStep + 1 TO GVL.A_LengthStep DO

    cmd := GVL_1.Step_Cr_A[i].Cmd;

    CASE cmd OF

        E_RobotCmd.CMD_IF,
        E_RobotCmd.CMD_IF_IN,
        E_RobotCmd.CMD_IF_VAR,
        E_RobotCmd.CMD_IF_REG:
            depth := depth + 1;


        E_RobotCmd.CMD_END_IF:
            IF depth = 0 THEN
                // Không có ELSE, nhảy tới sau END_IF
                F_FindElseOrEndIf_A := i + 1;
                RETURN;
            ELSE
                depth := depth - 1;
            END_IF;


        E_RobotCmd.CMD_ELSE:
            IF depth = 0 THEN
                // Có ELSE, nhảy tới step sau ELSE
                F_FindElseOrEndIf_A := i + 1;
                RETURN;
            END_IF;

    END_CASE;

END_FOR;

// Không tìm thấy thì báo về cuối chương trình
F_FindElseOrEndIf_A := GVL.A_LengthStep + 1;

END_FUNCTION

// Just_Motion_Control_x86_64_Linux_SM_WV/Application/FC_/RBA/F_CompareDINT_A
FUNCTION F_CompareDINT_A : BOOL
VAR_INPUT
	Actual   : DINT;
    Operator : DINT;
    SetValue : DINT;
END_VAR
VAR
END_VAR

CASE Operator OF
    1: F_CompareDINT_A := Actual =  SetValue;
    2: F_CompareDINT_A := Actual <> SetValue;
    3: F_CompareDINT_A := Actual >  SetValue;
    4: F_CompareDINT_A := Actual >= SetValue;
    5: F_CompareDINT_A := Actual <  SetValue;
    6: F_CompareDINT_A := Actual <= SetValue;
ELSE
    F_CompareDINT_A := FALSE;
END_CASE;

END_FUNCTION

// Just_Motion_Control_x86_64_Linux_SM_WV/Application/FC_/RBA/F_FindEndIf_A
FUNCTION F_FindEndIf_A : INT
VAR_INPUT
    StartStep : INT;
END_VAR

VAR
    i : INT;
    depth : INT;
    cmd : E_RobotCmd;
END_VAR

//====================================================
// Tìm END_IF tương ứng với ELSE hiện tại
// Có hỗ trợ IF lồng nhau
//====================================================

depth := 0;

FOR i := StartStep + 1 TO GVL.A_LengthStep DO

    cmd := GVL_1.Step_Cr_A[i].Cmd;

    CASE cmd OF

        E_RobotCmd.CMD_IF,
        E_RobotCmd.CMD_IF_IN,
        E_RobotCmd.CMD_IF_VAR,
        E_RobotCmd.CMD_IF_REG:
			// gặp IF con trong nhánh ELSE
            depth := depth + 1;


        E_RobotCmd.CMD_END_IF:
            IF depth = 0 THEN
                // Nhảy tới sau END_IF, END_IF tương ứng với ELSE hiện tại
                F_FindEndIf_A := i + 1;
                RETURN;
            ELSE
                depth := depth - 1;
            END_IF;

    END_CASE;

END_FOR;

F_FindEndIf_A := GVL.A_LengthStep + 1;

END_FUNCTION

// Just_Motion_Control_x86_64_Linux_SM_WV/Application/FC_/RBA/F_FindEndWhile_A
FUNCTION F_FindEndWhile_A : INT
VAR_INPUT
    StartStep : INT;
END_VAR

VAR
    i : INT;
    depth : INT;
    cmd : E_RobotCmd;
END_VAR

//====================================================
// Tìm END_WHILE tương ứng với WHILE tại StartStep
// Có hỗ trợ WHILE lồng nhau
//====================================================

depth := 0;

FOR i := StartStep + 1 TO GVL.A_LengthStep DO

    cmd := GVL_1.Step_Cr_A[i].Cmd;

    CASE cmd OF

        E_RobotCmd.CMD_WHILE,
        E_RobotCmd.CMD_WHILE_IN,
        E_RobotCmd.CMD_WHILE_REG:
            depth := depth + 1;


        E_RobotCmd.CMD_END_WHILE:
            IF depth = 0 THEN
                // WHILE sai, nhảy tới sau END_WHILE
                F_FindEndWhile_A := i + 1;
                RETURN;
            ELSE
                depth := depth - 1;
            END_IF;

    END_CASE;

END_FOR;

F_FindEndWhile_A := GVL.A_LengthStep + 1;

END_FUNCTION

// Just_Motion_Control_x86_64_Linux_SM_WV/Application/FC_/RBA/F_FindWhileStart_A
FUNCTION F_FindWhileStart_A : INT
VAR_INPUT
    EndWhileStep : INT;
END_VAR

VAR
    i : INT;
    depth : INT;
    cmd : E_RobotCmd;
END_VAR

//====================================================
// Tìm WHILE tương ứng khi đang đứng tại END_WHILE
// Quét ngược và hỗ trợ WHILE lồng nhau
//====================================================

depth := 0;

FOR i := EndWhileStep - 1 TO 1 BY -1 DO

    cmd := GVL_1.Step_Cr_A[i].Cmd;

    CASE cmd OF

        E_RobotCmd.CMD_END_WHILE:
            depth := depth + 1;


        E_RobotCmd.CMD_WHILE,
        E_RobotCmd.CMD_WHILE_IN,
        E_RobotCmd.CMD_WHILE_REG:
            IF depth = 0 THEN
                F_FindWhileStart_A := i;
                RETURN;
            ELSE
                depth := depth - 1;
            END_IF;

    END_CASE;

END_FOR;

F_FindWhileStart_A := 1;




// E_RobotCmd.CMD_ELSE:
//     // Nếu đã chạy nhánh IF TRUE, gặp ELSE thì bỏ qua ELSE block
//     GVL.A_RunStep := F_FindEndIf_A(GVL.A_RunStep);
//     GVL.A_RunState := 0;
// 

// E_RobotCmd.CMD_END_IF:
//     // Kết thúc IF block
//     GVL.A_RunStep := GVL.A_RunStep + 1;
//     GVL.A_RunState := 0;
// 
// 
// E_RobotCmd.CMD_WHILE:
//     // P1 = Condition No
//     IF F_EvalCondition_A(step_PRG_A_Interpreter.P1) THEN
//         GVL.A_RunStep := GVL.A_RunStep + 1;
//     ELSE
//         GVL.A_RunStep := F_FindEndWhile_A(GVL.A_RunStep);
//     END_IF;
// 
//     GVL.A_RunState := 0;
// 
// 
// E_RobotCmd.CMD_END_WHILE:
//     // Quay lại đầu WHILE để kiểm tra điều kiện lại
//     GVL.A_RunStep := F_FindWhileStart_A(GVL.A_RunStep);
//     GVL.A_RunState := 0;

END_FUNCTION

// Just_Motion_Control_x86_64_Linux_SM_WV/Application/FC_/RBA/F_CalcReg_A
FUNCTION F_CalcReg_A : DINT
VAR_INPUT
    Cmd       : E_RobotCmd;
    DestReg   : DINT;
    SourceMode: DINT;
    P3        : DINT;
    P4        : DINT;
END_VAR

VAR
    A : DINT;
    B : DINT;
END_VAR

//====================================================
// SourceMode:
// 0: RegDest với số cố định P3
// 1: RegDest với Reg[P3]
// 2: Reg[P3] với Reg[P4], trả về RegDest
//====================================================

IF (DestReg < 1) OR (DestReg > 200) THEN
    F_CalcReg_A := 0;
    RETURN;
END_IF;

CASE SourceMode OF

    0:
        A := GVL.A_Reg[DestReg];
        B := P3;

    1:
        A := GVL.A_Reg[DestReg];

        IF (P3 >= 1) AND (P3 <= 200) THEN
            B := GVL.A_Reg[P3];
        ELSE
            B := 0;
        END_IF;

    2:
        IF (P3 >= 1) AND (P3 <= 200) THEN
            A := GVL.A_Reg[P3];
        ELSE
            A := 0;
        END_IF;

        IF (P4 >= 1) AND (P4 <= 200) THEN
            B := GVL.A_Reg[P4];
        ELSE
            B := 0;
        END_IF;

ELSE
    A := GVL.A_Reg[DestReg];
    B := 0;

END_CASE;


CASE Cmd OF

    E_RobotCmd.CMD_REG_SET:
        F_CalcReg_A := B;

    E_RobotCmd.CMD_REG_ADD:
        F_CalcReg_A := A + B;

    E_RobotCmd.CMD_REG_SUB:
        F_CalcReg_A := A - B;

    E_RobotCmd.CMD_REG_MUL:
        F_CalcReg_A := A * B;

    E_RobotCmd.CMD_REG_DIV:
        IF B <> 0 THEN
            F_CalcReg_A := A / B;
        ELSE
            F_CalcReg_A := GVL.A_Reg[DestReg];
        END_IF;

    E_RobotCmd.CMD_REG_MOD:
        IF B <> 0 THEN
            F_CalcReg_A := A MOD B;
        ELSE
            F_CalcReg_A := GVL.A_Reg[DestReg];
        END_IF;

ELSE
    F_CalcReg_A := GVL.A_Reg[DestReg];

END_CASE;

END_FUNCTION

// Just_Motion_Control_x86_64_Linux_SM_WV/Application/FC_/RBA/F_CalcVar_A
FUNCTION F_CalcVar_A : DINT
VAR_INPUT
    Cmd        : E_RobotCmd;
    DestVar    : DINT;
    SourceMode : DINT;
    P3         : DINT;
    P4         : DINT;
END_VAR

VAR
    A : DINT;
    B : DINT;
END_VAR

IF (DestVar < 1) OR (DestVar > 200) THEN
    F_CalcVar_A := 0;
    RETURN;
END_IF;

CASE SourceMode OF
    0: // VarDest với số cố định P3
        A := GVL.A_Var[DestVar];
        B := P3;

    1: // VarDest với Var[P3]
        A := GVL.A_Var[DestVar];

        IF (P3 >= 1) AND (P3 <= 200) THEN
            B := GVL.A_Var[P3];
        ELSE
            B := 0;
        END_IF;

    2: // Var[P3] với Var[P4], trả về VarDest
        IF (P3 >= 1) AND (P3 <= 200) THEN
            A := GVL.A_Var[P3];
        ELSE
            A := 0;
        END_IF;

        IF (P4 >= 1) AND (P4 <= 200) THEN
            B := GVL.A_Var[P4];
        ELSE
            B := 0;
        END_IF;
ELSE
    A := GVL.A_Var[DestVar];
    B := 0;
END_CASE;

CASE Cmd OF
    E_RobotCmd.CMD_VAR_SET:
        F_CalcVar_A := B;

    E_RobotCmd.CMD_VAR_ADD:
        F_CalcVar_A := A + B;

    E_RobotCmd.CMD_VAR_SUB:
        F_CalcVar_A := A - B;

    E_RobotCmd.CMD_VAR_MUL:
        F_CalcVar_A := A * B;

    E_RobotCmd.CMD_VAR_DIV:
        IF B <> 0 THEN
            F_CalcVar_A := A / B;
        ELSE
            F_CalcVar_A := GVL.A_Var[DestVar];
        END_IF;

    E_RobotCmd.CMD_VAR_MOD:
        IF B <> 0 THEN
            F_CalcVar_A := A MOD B;
        ELSE
            F_CalcVar_A := GVL.A_Var[DestVar];
        END_IF;

ELSE
    F_CalcVar_A := GVL.A_Var[DestVar];
END_CASE;

END_FUNCTION

// Just_Motion_Control_x86_64_Linux_SM_WV/Application/FC_/F_BuildMotionItem
FUNCTION F_BuildMotionItem  : ST_MotionQueueItem // Tao motion item dua vào queue
VAR_INPUT
	StepNo : INT;
END_VAR
VAR
	Step    : ST_RobotStep;
    item : ST_MotionQueueItem;
END_VAR

// Lấy dữ liệu Step hiện tại
Step := GVL_1.Step_Cr_A[StepNo];

// Xóa dữ liệu cũ trong item
item.Cmd        := Step.Cmd;
item.SourceStep := StepNo;
item.PointNo    := 0;
item.MidPointNo := 0;
item.EndPointNo := 0;
item.Speed      := 0.0;
item.BlendMode  := 0;
item.BlendRadius := 0.0;
item.CircleMode := 0;
item.PathChoice := 0;
item.SkipPositionCheck := FALSE;

// Phân tích theo từng loại lệnh Motion
CASE Step.Cmd OF

    // MovP / MovL
    E_RobotCmd.CMD_MovP,
    E_RobotCmd.CMD_MovL:

        // P1 = Point No
        item.PointNo := Step.P1;

        // P2 = Speed override
        // Nếu P2 = 0 thì FB sẽ dùng tốc độ từ Set Speed
        IF Step.P2 > 0 THEN
            item.Speed := INT_TO_LREAL(Step.P2);
        END_IF;

        // P3 = BlendMode
        // 0=None, 1=TMCornerDistance, 2=TMStartVelocity
        item.BlendMode := TO_INT(Step.P3);

        // P4 = BlendRadius
        item.BlendRadius := INT_TO_LREAL(Step.P4);
		IF F_IsMotionCmd(GVL_1.Step_Cr_A[StepNo + 1].Cmd) AND (GVL_1.Step_Cr_A[StepNo + 1].P3 >0) THEN
			item.SkipPositionCheck := TRUE;
		END_IF

    // MovC
    E_RobotCmd.CMD_MovC:

        // P1 = Mid Point
        item.MidPointNo := Step.P1;

        // P2 = End Point
        item.EndPointNo := Step.P2;

        // P3 = CircleMode
        item.CircleMode := TO_INT(Step.P3);

        // P4 = PathChoice
        item.PathChoice := Step.P4;

        // P5 = Speed override
        IF Step.P5 > 0 THEN
            item.Speed := INT_TO_LREAL(Step.P5);
        END_IF;
		
		IF F_IsMotionCmd(GVL_1.Step_Cr_A[StepNo + 1].Cmd) AND (GVL_1.Step_Cr_A[StepNo + 1].P3 >0) THEN
			item.SkipPositionCheck := TRUE;
		END_IF

END_CASE;

// Trả item cho Motion Queue
F_BuildMotionItem := item;

END_FUNCTION

// Just_Motion_Control_x86_64_Linux_SM_WV/Application/FC_/F_GetFreeMoveSlot
FUNCTION F_GetFreeMoveSlot  : INT // Tra lai Slot Free Cua cac ham motion
VAR_INPUT
END_VAR
VAR
	i : INT;
END_VAR

F_GetFreeMoveSlot := 0;

FOR i := 1 TO 3 DO
    IF NOT GVL.A_MoveSlotBusy[i] AND NOT GVL.A_MoveSlotDone[i] AND NOT GVL.A_MoveSlotAccepted[i] THEN
        F_GetFreeMoveSlot := i;
        RETURN;
    END_IF;
END_FOR;

END_FUNCTION

// Just_Motion_Control_x86_64_Linux_SM_WV/Application/FC_/RBA/F_GetPointSMC_A
FUNCTION F_GetPointSMC_A  : SMC_POS_REF
VAR_INPUT
	PointNo : INT;
END_VAR
VAR
	pos : SMC_POS_REF;
END_VAR

//====================================================
// F_GetPointSMC_A
// Chuyển dữ liệu điểm dạng mảng X/Y/Z/A của anh
// sang kiểu SMC_POS_REF để đưa vào FB Motion
//====================================================

// Kiểm tra giới hạn point
IF (PointNo < 1) OR (PointNo > 500) THEN
    // Nếu lỗi point thì trả về điểm 0
    // Lỗi thật nên bắt thêm ở Build/Run sau
    F_GetPointSMC_A := pos;
    RETURN;
END_IF;

// Gán tọa độ Cartesian
pos.c.X := GVL_1.DATA_RB_A.X_POS[PointNo]; // X
pos.c.Y := GVL_1.DATA_RB_A.Y_POS[PointNo]; // Y
pos.c.Z := GVL_1.DATA_RB_A.Z_POS[PointNo]; // Z

// Với SCARA thường A là góc quay quanh Z
// Tùy cấu hình robot, A có thể là c[3] hoặc orientation field khác
pos.c.A := GVL_1.DATA_RB_A.R_POS[PointNo]; // A / Rz

// Trả kết quả
F_GetPointSMC_A := pos;

END_FUNCTION

// Just_Motion_Control_x86_64_Linux_SM_WV/Application/FC_/RBB/F_EvalCondition_B
FUNCTION F_EvalCondition_B : BOOL
VAR_INPUT
    CondNo : INT;
END_VAR
VAR
    i : INT;
    rowResult : BOOL;
    finalResult : BOOL;
    firstRow : BOOL;
END_VAR

// IMPLEMENTATION
IF (CondNo < 1) OR (CondNo > 100) THEN
    F_EvalCondition_B := FALSE;
    RETURN;
END_IF;

IF NOT GVL_1.Condition_Cr_B[CondNo].Enable THEN
    F_EvalCondition_B := FALSE;
    RETURN;
END_IF;

firstRow := TRUE;
finalResult := FALSE;

FOR i := 1 TO 10 DO

    IF GVL_1.Condition_Cr_B[CondNo].Row[i].Enable THEN

        rowResult := F_EvalCondRow_B(GVL_1.Condition_Cr_B[CondNo].Row[i]);

        IF firstRow THEN
            finalResult := rowResult;
            firstRow := FALSE;
        ELSE
            CASE GVL_1.Condition_Cr_B[CondNo].Row[i - 1].LinkNext OF
                1: finalResult := finalResult AND rowResult;
                2: finalResult := finalResult OR rowResult;
            ELSE
                finalResult := finalResult AND rowResult;
            END_CASE;
        END_IF;

    END_IF;

END_FOR;

GVL_1.Condition_Cr_B[CondNo].Result := finalResult;
F_EvalCondition_B := finalResult;

END_FUNCTION

// Just_Motion_Control_x86_64_Linux_SM_WV/Application/FC_/RBB/F_EvalCondRow_B
FUNCTION F_EvalCondRow_B : BOOL
VAR_INPUT
    Row : ST_ConditionRow;
END_VAR
VAR
    actualValue : LREAL;
END_VAR

// IMPLEMENTATION
IF NOT Row.Enable THEN
    F_EvalCondRow_B := TRUE;
    RETURN;
END_IF;

actualValue := F_GetCondValue_B(
    Source := Row.Source,
    Index  := Row.Index
);

CASE Row.Operator OF
    1: F_EvalCondRow_B := actualValue = Row.SetValue;
    2: F_EvalCondRow_B := actualValue <> Row.SetValue;
    3: F_EvalCondRow_B := actualValue > Row.SetValue;
    4: F_EvalCondRow_B := actualValue >= Row.SetValue;
    5: F_EvalCondRow_B := actualValue < Row.SetValue;
    6: F_EvalCondRow_B := actualValue <= Row.SetValue;
ELSE
    F_EvalCondRow_B := FALSE;
END_CASE;

END_FUNCTION

// Just_Motion_Control_x86_64_Linux_SM_WV/Application/FC_/RBB/F_GetCondValue_B
FUNCTION F_GetCondValue_B : DINT
VAR_INPUT
    Source : INT;
    Index : INT;
END_VAR

// IMPLEMENTATION
CASE Source OF
	0:
    1: // DI
        IF GVL.X[Index] THEN
            F_GetCondValue_B := 1;
        ELSE
            F_GetCondValue_B := 0;
        END_IF;

    2: // DO
        IF GVL.Y[Index] THEN
            F_GetCondValue_B := 1;
        ELSE
            F_GetCondValue_B := 0;
        END_IF;

//     3: // REG
//         F_GetCondValue_B := GVL.B_Reg[Index];
// 
//     4: // VAR
//         F_GetCondValue_B := GVL.B_Var[Index];

ELSE
    F_GetCondValue_B := 0;

END_CASE;

END_FUNCTION

// Just_Motion_Control_x86_64_Linux_SM_WV/Application/FC_/RBB/F_FindElseOrEndIf_B
FUNCTION F_FindElseOrEndIf_B : INT
VAR_INPUT
    StartStep : INT;
END_VAR
VAR
    i : INT;
    depth : INT;
    cmd : E_RobotCmd;
END_VAR

// IMPLEMENTATION
//====================================================
// Tìm ELSE hoặc END_IF tương ứng với IF tại StartStep
// Có hỗ trợ IF lồng nhau
//====================================================

depth := 0;

FOR i := StartStep + 1 TO GVL.B_LengthStep DO

    cmd := GVL_1.Step_Cr_B[i].Cmd;

    CASE cmd OF

        E_RobotCmd.CMD_IF,
        E_RobotCmd.CMD_IF_IN,
        E_RobotCmd.CMD_IF_VAR,
        E_RobotCmd.CMD_IF_REG:
            depth := depth + 1;


        E_RobotCmd.CMD_END_IF:
            IF depth = 0 THEN
                // Không có ELSE, nhảy tới sau END_IF
                F_FindElseOrEndIf_B := i + 1;
                RETURN;
            ELSE
                depth := depth - 1;
            END_IF;


        E_RobotCmd.CMD_ELSE:
            IF depth = 0 THEN
                // Có ELSE, nhảy tới step sau ELSE
                F_FindElseOrEndIf_B := i + 1;
                RETURN;
            END_IF;

    END_CASE;

END_FOR;

// Không tìm thấy thì báo về cuối chương trình
F_FindElseOrEndIf_B := GVL.B_LengthStep + 1;

END_FUNCTION

// Just_Motion_Control_x86_64_Linux_SM_WV/Application/FC_/RBB/F_CompareDINT_B
FUNCTION F_CompareDINT_B : BOOL
VAR_INPUT
    Actual : DINT;
    Operator : DINT;
    SetValue : DINT;
END_VAR

// IMPLEMENTATION
CASE Operator OF
    1: F_CompareDINT_B := Actual =  SetValue;
    2: F_CompareDINT_B := Actual <> SetValue;
    3: F_CompareDINT_B := Actual >  SetValue;
    4: F_CompareDINT_B := Actual >= SetValue;
    5: F_CompareDINT_B := Actual <  SetValue;
    6: F_CompareDINT_B := Actual <= SetValue;
ELSE
    F_CompareDINT_B := FALSE;
END_CASE;

END_FUNCTION

// Just_Motion_Control_x86_64_Linux_SM_WV/Application/FC_/RBB/F_FindEndIf_B
FUNCTION F_FindEndIf_B : INT
VAR_INPUT
    StartStep : INT;
END_VAR
VAR
    i : INT;
    depth : INT;
    cmd : E_RobotCmd;
END_VAR

// IMPLEMENTATION
//====================================================
// Tìm END_IF tương ứng với ELSE hiện tại
// Có hỗ trợ IF lồng nhau
//====================================================

depth := 0;

FOR i := StartStep + 1 TO GVL.B_LengthStep DO

    cmd := GVL_1.Step_Cr_B[i].Cmd;

    CASE cmd OF

        E_RobotCmd.CMD_IF,
        E_RobotCmd.CMD_IF_IN,
        E_RobotCmd.CMD_IF_VAR,
        E_RobotCmd.CMD_IF_REG:
			// gặp IF con trong nhánh ELSE
            depth := depth + 1;


        E_RobotCmd.CMD_END_IF:
            IF depth = 0 THEN
                // Nhảy tới sau END_IF, END_IF tương ứng với ELSE hiện tại
                F_FindEndIf_B := i + 1;
                RETURN;
            ELSE
                depth := depth - 1;
            END_IF;

    END_CASE;

END_FOR;

F_FindEndIf_B := GVL.B_LengthStep + 1;

END_FUNCTION

// Just_Motion_Control_x86_64_Linux_SM_WV/Application/FC_/RBB/F_FindEndWhile_B
FUNCTION F_FindEndWhile_B : INT
VAR_INPUT
    StartStep : INT;
END_VAR
VAR
    i : INT;
    depth : INT;
    cmd : E_RobotCmd;
END_VAR

// IMPLEMENTATION
//====================================================
// Tìm END_WHILE tương ứng với WHILE tại StartStep
// Có hỗ trợ WHILE lồng nhau
//====================================================

depth := 0;

FOR i := StartStep + 1 TO GVL.B_LengthStep DO

    cmd := GVL_1.Step_Cr_B[i].Cmd;

    CASE cmd OF

        E_RobotCmd.CMD_WHILE,
        E_RobotCmd.CMD_WHILE_IN,
        E_RobotCmd.CMD_WHILE_REG:
            depth := depth + 1;


        E_RobotCmd.CMD_END_WHILE:
            IF depth = 0 THEN
                // WHILE sai, nhảy tới sau END_WHILE
                F_FindEndWhile_B := i + 1;
                RETURN;
            ELSE
                depth := depth - 1;
            END_IF;

    END_CASE;

END_FOR;

F_FindEndWhile_B := GVL.B_LengthStep + 1;

END_FUNCTION

// Just_Motion_Control_x86_64_Linux_SM_WV/Application/FC_/RBB/F_FindWhileStart_B
FUNCTION F_FindWhileStart_B : INT
VAR_INPUT
    EndWhileStep : INT;
END_VAR
VAR
    i : INT;
    depth : INT;
    cmd : E_RobotCmd;
END_VAR

// IMPLEMENTATION
//====================================================
// Tìm WHILE tương ứng khi đang đứng tại END_WHILE
// Quét ngược và hỗ trợ WHILE lồng nhau
//====================================================

depth := 0;

FOR i := EndWhileStep - 1 TO 1 BY -1 DO

    cmd := GVL_1.Step_Cr_B[i].Cmd;

    CASE cmd OF

        E_RobotCmd.CMD_END_WHILE:
            depth := depth + 1;


        E_RobotCmd.CMD_WHILE,
        E_RobotCmd.CMD_WHILE_IN,
        E_RobotCmd.CMD_WHILE_REG:
            IF depth = 0 THEN
                F_FindWhileStart_B := i;
                RETURN;
            ELSE
                depth := depth - 1;
            END_IF;

    END_CASE;

END_FOR;

F_FindWhileStart_B := 1;




// E_RobotCmd.CMD_ELSE:
//     // Nếu đã chạy nhánh IF TRUE, gặp ELSE thì bỏ qua ELSE block
//     GVL.A_RunStep := F_FindEndIf_B(GVL.A_RunStep);
//     GVL.A_RunState := 0;
// 

// E_RobotCmd.CMD_END_IF:
//     // Kết thúc IF block
//     GVL.A_RunStep := GVL.A_RunStep + 1;
//     GVL.A_RunState := 0;
// 
// 
// E_RobotCmd.CMD_WHILE:
//     // P1 = Condition No
//     IF F_EvalCondition_B(step_PRG_A_Interpreter.P1) THEN
//         GVL.A_RunStep := GVL.A_RunStep + 1;
//     ELSE
//         GVL.A_RunStep := F_FindEndWhile_B(GVL.A_RunStep);
//     END_IF;
// 
//     GVL.A_RunState := 0;
// 
// 
// E_RobotCmd.CMD_END_WHILE:
//     // Quay lại đầu WHILE để kiểm tra điều kiện lại
//     GVL.A_RunStep := F_FindWhileStart_B(GVL.A_RunStep);
//     GVL.A_RunState := 0;

END_FUNCTION

// Just_Motion_Control_x86_64_Linux_SM_WV/Application/FC_/RBB/F_CalcReg_B
FUNCTION F_CalcReg_B : DINT
VAR_INPUT
    Cmd : E_RobotCmd;
    DestReg : DINT;
    SourceMode : DINT;
    P3 : DINT;
    P4 : DINT;
END_VAR
VAR
    A : DINT;
    B : DINT;
END_VAR

// IMPLEMENTATION
//====================================================
// SourceMode:
// 0: RegDest với số cố định P3
// 1: RegDest với Reg[P3]
// 2: Reg[P3] với Reg[P4], trả về RegDest
//====================================================

IF (DestReg < 1) OR (DestReg > 200) THEN
    F_CalcReg_B := 0;
    RETURN;
END_IF;

CASE SourceMode OF

    0:
        A := GVL.B_Reg[DestReg];
        B := P3;

    1:
        A := GVL.B_Reg[DestReg];

        IF (P3 >= 1) AND (P3 <= 200) THEN
            B := GVL.B_Reg[P3];
        ELSE
            B := 0;
        END_IF;

    2:
        IF (P3 >= 1) AND (P3 <= 200) THEN
            A := GVL.B_Reg[P3];
        ELSE
            A := 0;
        END_IF;

        IF (P4 >= 1) AND (P4 <= 200) THEN
            B := GVL.B_Reg[P4];
        ELSE
            B := 0;
        END_IF;

ELSE
    A := GVL.B_Reg[DestReg];
    B := 0;

END_CASE;


CASE Cmd OF

    E_RobotCmd.CMD_REG_SET:
        F_CalcReg_B := B;

    E_RobotCmd.CMD_REG_ADD:
        F_CalcReg_B := A + B;

    E_RobotCmd.CMD_REG_SUB:
        F_CalcReg_B := A - B;

    E_RobotCmd.CMD_REG_MUL:
        F_CalcReg_B := A * B;

    E_RobotCmd.CMD_REG_DIV:
        IF B <> 0 THEN
            F_CalcReg_B := A / B;
        ELSE
            F_CalcReg_B := GVL.B_Reg[DestReg];
        END_IF;

    E_RobotCmd.CMD_REG_MOD:
        IF B <> 0 THEN
            F_CalcReg_B := A MOD B;
        ELSE
            F_CalcReg_B := GVL.B_Reg[DestReg];
        END_IF;

ELSE
    F_CalcReg_B := GVL.B_Reg[DestReg];

END_CASE;

END_FUNCTION

// Just_Motion_Control_x86_64_Linux_SM_WV/Application/FC_/RBB/F_CalcVar_B
FUNCTION F_CalcVar_B : DINT
VAR_INPUT
    Cmd : E_RobotCmd;
    DestVar : DINT;
    SourceMode : DINT;
    P3 : DINT;
    P4 : DINT;
END_VAR
VAR
    A : DINT;
    B : DINT;
END_VAR

// IMPLEMENTATION
IF (DestVar < 1) OR (DestVar > 200) THEN
    F_CalcVar_B := 0;
    RETURN;
END_IF;

CASE SourceMode OF
    0: // VarDest với số cố định P3
        A := GVL.B_Var[DestVar];
        B := P3;

    1: // VarDest với Var[P3]
        A := GVL.B_Var[DestVar];

        IF (P3 >= 1) AND (P3 <= 200) THEN
            B := GVL.B_Var[P3];
        ELSE
            B := 0;
        END_IF;

    2: // Var[P3] với Var[P4], trả về VarDest
        IF (P3 >= 1) AND (P3 <= 200) THEN
            A := GVL.B_Var[P3];
        ELSE
            A := 0;
        END_IF;

        IF (P4 >= 1) AND (P4 <= 200) THEN
            B := GVL.B_Var[P4];
        ELSE
            B := 0;
        END_IF;
ELSE
    A := GVL.B_Var[DestVar];
    B := 0;
END_CASE;

CASE Cmd OF
    E_RobotCmd.CMD_VAR_SET:
        F_CalcVar_B := B;

    E_RobotCmd.CMD_VAR_ADD:
        F_CalcVar_B := A + B;

    E_RobotCmd.CMD_VAR_SUB:
        F_CalcVar_B := A - B;

    E_RobotCmd.CMD_VAR_MUL:
        F_CalcVar_B := A * B;

    E_RobotCmd.CMD_VAR_DIV:
        IF B <> 0 THEN
            F_CalcVar_B := A / B;
        ELSE
            F_CalcVar_B := GVL.B_Var[DestVar];
        END_IF;

    E_RobotCmd.CMD_VAR_MOD:
        IF B <> 0 THEN
            F_CalcVar_B := A MOD B;
        ELSE
            F_CalcVar_B := GVL.B_Var[DestVar];
        END_IF;

ELSE
    F_CalcVar_B := GVL.B_Var[DestVar];
END_CASE;

END_FUNCTION

// Just_Motion_Control_x86_64_Linux_SM_WV/Application/FC_/F_BuildMotionItem_B
FUNCTION F_BuildMotionItem_B  : ST_MotionQueueItem // Tao motion item dua vào queue
VAR_INPUT
	StepNo : INT;
END_VAR
VAR
	Step    : ST_RobotStep;
    item : ST_MotionQueueItem;
END_VAR

// Lấy dữ liệu Step hiện tại
Step := GVL_1.Step_Cr_B[StepNo];

// Xóa dữ liệu cũ trong item
item.Cmd        := Step.Cmd;
item.SourceStep := StepNo;
item.PointNo    := 0;
item.MidPointNo := 0;
item.EndPointNo := 0;
item.Speed      := 0.0;
item.BlendMode  := 0;
item.BlendRadius := 0.0;
item.CircleMode := 0;
item.PathChoice := 0;
item.SkipPositionCheck := FALSE;

// Phân tích theo từng loại lệnh Motion
CASE Step.Cmd OF

    // MovP / MovL
    E_RobotCmd.CMD_MovP,
    E_RobotCmd.CMD_MovL:

        // P1 = Point No
        item.PointNo := Step.P1;

        // P2 = Speed override
        // Nếu P2 = 0 thì FB sẽ dùng tốc độ từ Set Speed
        IF Step.P2 > 0 THEN
            item.Speed := INT_TO_LREAL(Step.P2);
        END_IF;

        // P3 = BlendMode
        // 0=None, 1=TMCornerDistance, 2=TMStartVelocity
        item.BlendMode := TO_INT(Step.P3);

        // P4 = BlendRadius
        item.BlendRadius := INT_TO_LREAL(Step.P4);
		IF F_IsMotionCmd(GVL_1.Step_Cr_B[StepNo + 1].Cmd) AND (GVL_1.Step_Cr_B[StepNo + 1].P3 >0) THEN
			item.SkipPositionCheck := TRUE;
		END_IF

    // MovC
    E_RobotCmd.CMD_MovC:

        // P1 = Mid Point
        item.MidPointNo := Step.P1;

        // P2 = End Point
        item.EndPointNo := Step.P2;

        // P3 = CircleMode
        item.CircleMode := TO_INT(Step.P3);

        // P4 = PathChoice
        item.PathChoice := Step.P4;

        // P5 = Speed override
        IF Step.P5 > 0 THEN
            item.Speed := INT_TO_LREAL(Step.P5);
        END_IF;
		
		IF F_IsMotionCmd(GVL_1.Step_Cr_B[StepNo + 1].Cmd) AND (GVL_1.Step_Cr_B[StepNo + 1].P3 >0) THEN
			item.SkipPositionCheck := TRUE;
		END_IF

END_CASE;

// Trả item cho Motion Queue
F_BuildMotionItem_B := item;

END_FUNCTION

// Just_Motion_Control_x86_64_Linux_SM_WV/Application/FC_/F_GetFreeMoveSlot_B
FUNCTION F_GetFreeMoveSlot_B  : INT // Tra lai Slot Free Cua cac ham motion
VAR_INPUT
END_VAR
VAR
	i : INT;
END_VAR

F_GetFreeMoveSlot_B := 0;

FOR i := 1 TO 3 DO
    IF NOT GVL.B_MoveSlotBusy[i] AND NOT GVL.B_MoveSlotDone[i] AND NOT GVL.B_MoveSlotAccepted[i] THEN
        F_GetFreeMoveSlot_B := i;
        RETURN;
    END_IF;
END_FOR;

END_FUNCTION

// Just_Motion_Control_x86_64_Linux_SM_WV/Application/FC_/RBB/F_GetPointSMC_B
FUNCTION F_GetPointSMC_B : SMC_POS_REF
VAR_INPUT
    PointNo : INT;
END_VAR
VAR
    pos : SMC_POS_REF;
END_VAR

// IMPLEMENTATION
//====================================================
// F_GetPointSMC_B
// Chuyển dữ liệu điểm dạng mảng X/Y/Z/A của anh
// sang kiểu SMC_POS_REF để đưa vào FB Motion
//====================================================

// Kiểm tra giới hạn point
IF (PointNo < 1) OR (PointNo > 500) THEN
    // Nếu lỗi point thì trả về điểm 0
    // Lỗi thật nên bắt thêm ở Build/Run sau
    F_GetPointSMC_B := pos;
    RETURN;
END_IF;

// Gán tọa độ Cartesian
pos.c.X := GVL_1.DATA_RB_B.X_POS[PointNo]; // X
pos.c.Y := GVL_1.DATA_RB_B.Y_POS[PointNo]; // Y
pos.c.Z := GVL_1.DATA_RB_B.Z_POS[PointNo]; // Z

// Với SCARA thường A là góc quay quanh Z
// Tùy cấu hình robot, A có thể là c[3] hoặc orientation field khác
pos.c.A := GVL_1.DATA_RB_B.R_POS[PointNo]; // A / Rz

// Trả kết quả
F_GetPointSMC_B := pos;

END_FUNCTION

// Just_Motion_Control_x86_64_Linux_SM_WV/Application/PRG_MACHINE/Monitor_Production
PROGRAM Monitor_Production
VAR_INPUT
	Pulse_In, Pulse_In_1, Pulse_In_2, Pulse_In_     : BOOL;
	Pulse_Out, Pulse_Out_1, Pulse_Out_2, Pulse_Out_     : BOOL;
    Pulse_Old, Pulse_Old_1, Pulse_Old_2, Pulse_Old_    : BOOL;
END_VAR
VAR
// Production Count
	D_Day_Pro, D_Night_Pro : ARRAY[0..11] OF WORD;
	D_Day_Pro_OK, D_Night_Pro_OK : ARRAY[0..11] OF WORD;
	Total_Day, Total_Night, All_Shift : WORD;
	i_qty : WORD;
	i : WORD;
	In_Qty, In_Qty_old : BOOL;
	In_Qty_NG_VS, In_Qty_old_NG_VS : BOOL;
	In_Qty_NG_TS, In_Qty_old_NG_TS : BOOL;
	Second, minute, hour, day, month, year : WORD;
	day_old : WORD;
	Clear_all, Shift_Reset_Day, Shift_Reset_Night, Shift_Reset_Day_Old, Shift_Reset_Night_Old : BOOL;
/// tactime
   
    // thời gian (ms)
	Tact_ms, Tact_ms_1, Tact_ms_2, Tact_ms_      : DWORD;   // giá trị ms để đưa ra HMI
	T1,T2,T3,T4           : TON;
    // buffer 10 lần
    Tact_Array,Tact_Array_1, Tact_Array_2, Tact_Array_   : ARRAY[0..9] OF WORD;
    Index, Index_1, Index_2, Index_,
	Count, Count_1, Count_2, Count_        : INT := 0;

    Avg_Tact, Avg_Tact_1, Avg_Tact_2, Avg_Tact_    : WORD;

    i_tactime_input,i_tactime_input_1,i_tactime_input_2, i_tactime_input_            : INT;
    Sum_Tact, Sum_Tact_1, Sum_Tact_2, Sum_Tact_    : WORD;	
	Clear_data_tacttime :BOOL;
	
END_VAR

/// Update Date
Second := GVL.DW_[30];
minute := GVL.DW_[31];
hour := GVL.DW_[32];
day := GVL.DW_[33];
month := GVL.DW_[34];
year := GVL.DW_[35];

///
Qty_Production();
Tactime_Input();
Tactime_MC1();
Tactime_MC2();
Tactime_output();
// 
IF Clear_data_tacttime THEN
	FOR i := 0 TO 9 DO
		Tact_Array[i] := 0;
		Tact_Array_1[i] := 0;
		Tact_Array_2[i] := 0;
		Tact_Array_[i] := 0;
	END_FOR
END_IF

ACTION Qty_Production:
// In_Qty := GVL.Pro4_.Signal_In.T_Cv_In_1.q;
In_Qty := (POU_MOTION.Pro_A4 = 80);
In_Qty_NG_VS := (POU_MOTION.Pro_A4 = 90);
In_Qty_NG_TS := (POU_MOTION.Pro_A4 = 100);
// Reset 08:00
Shift_Reset_Day := (hour = 8) AND (minute = 0);

// Reset 20:00
Shift_Reset_Night := (hour = 20) AND (minute = 0);

// ===== RESET day shift =====
IF  ( (Shift_Reset_Day = TRUE) AND (Shift_Reset_Day_Old = FALSE) ) OR Clear_all THEN
    FOR i := 0 TO 11 DO
        GVL.Pro4_.Monitor.D_Day_Pro_OK[i] := 0;
		GVL.Pro4_.Monitor.D_Day_Pro_NG_VS[i] := 0;
		GVL.Pro4_.Monitor.D_Day_Pro_NG_TS[i] := 0;
    END_FOR
END_IF
Shift_Reset_Day_Old := Shift_Reset_Day;


// ===== RESET night shift =====
IF ((Shift_Reset_Night = TRUE) AND (Shift_Reset_Night_Old = FALSE)) OR Clear_all THEN
    FOR i := 0 TO 11 DO
        GVL.Pro4_.Monitor.D_Night_Pro_OK[i] := 0;
		GVL.Pro4_.Monitor.D_Night_Pro_NG_VS[i] := 0;
		GVL.Pro4_.Monitor.D_Night_Pro_NG_TS[i] := 0;
    END_FOR
END_IF
Shift_Reset_Night_Old := Shift_Reset_Night;		

/// counter OK
IF (In_Qty = TRUE) AND (In_Qty_old = FALSE) THEN

    // 8h -> 19h 
    IF (hour >= 8) AND (hour < 20) THEN
        GVL.Pro4_.Monitor.D_Day_Pro_OK[hour - 8] := GVL.Pro4_.Monitor.D_Day_Pro_OK[hour - 8] + 1;
    END_IF

    // 20h -> 7h 
    IF (hour >= 20) THEN
        GVL.Pro4_.Monitor.D_Night_Pro_OK[hour - 20] := GVL.Pro4_.Monitor.D_Night_Pro_OK[hour - 20] + 1;
    ELSIF (hour < 8) THEN
        GVL.Pro4_.Monitor.D_Night_Pro_OK[hour + 4] := GVL.Pro4_.Monitor.D_Night_Pro_OK[hour + 4] + 1;
    END_IF

END_IF
In_Qty_old := In_Qty;

/// counter NG_VS
IF (In_Qty_NG_VS = TRUE) AND (In_Qty_old_NG_VS = FALSE) THEN

    // 8h -> 19h 
    IF (hour >= 8) AND (hour < 20) THEN
        GVL.Pro4_.Monitor.D_Day_Pro_NG_VS[hour - 8] := GVL.Pro4_.Monitor.D_Day_Pro_NG_VS[hour - 8] + 1;
    END_IF

    // 20h -> 7h 
    IF (hour >= 20) THEN
        GVL.Pro4_.Monitor.D_Night_Pro_NG_VS[hour - 20] := GVL.Pro4_.Monitor.D_Night_Pro_NG_VS[hour - 20] + 1;
    ELSIF (hour < 8) THEN
        GVL.Pro4_.Monitor.D_Night_Pro_NG_VS[hour + 4] := GVL.Pro4_.Monitor.D_Night_Pro_NG_VS[hour + 4] + 1;
    END_IF

END_IF
In_Qty_old_NG_VS := In_Qty_NG_VS;

/// counter NG_TS
IF (In_Qty_NG_TS = TRUE) AND (In_Qty_old_NG_TS = FALSE) THEN

    // 8h -> 19h 
    IF (hour >= 8) AND (hour < 20) THEN
        GVL.Pro4_.Monitor.D_Day_Pro_NG_TS[hour - 8] := GVL.Pro4_.Monitor.D_Day_Pro_NG_TS[hour - 8] + 1;
    END_IF

    // 20h -> 7h 
    IF (hour >= 20) THEN
        GVL.Pro4_.Monitor.D_Night_Pro_NG_TS[hour - 20] := GVL.Pro4_.Monitor.D_Night_Pro_NG_TS[hour - 20] + 1;
    ELSIF (hour < 8) THEN
        GVL.Pro4_.Monitor.D_Night_Pro_NG_TS[hour + 4] := GVL.Pro4_.Monitor.D_Night_Pro_NG_TS[hour + 4] + 1;
    END_IF

END_IF
In_Qty_old_NG_TS := In_Qty_NG_TS;

/// Total Production
// GVL.Pro4_.Monitor.Total_Day := 0;
// GVL.Pro4_.Monitor.Total_Night := 0;
GVL.Pro4_.Monitor.Total_Day_OK := 0;
GVL.Pro4_.Monitor.Total_Night_OK := 0;
GVL.Pro4_.Monitor.Total_Day_NG_VS := 0;
GVL.Pro4_.Monitor.Total_Night_NG_VS := 0;
GVL.Pro4_.Monitor.Total_Day_NG_TS := 0;
GVL.Pro4_.Monitor.Total_Night_NG_TS := 0;

FOR i_qty := 0 TO 11 BY 1 DO
	GVL.Pro4_.Monitor.Total_Day_OK := GVL.Pro4_.Monitor.Total_Day_OK + GVL.Pro4_.Monitor.D_Day_Pro_OK[i_qty];
	GVL.Pro4_.Monitor.Total_Night_OK := GVL.Pro4_.Monitor.Total_Night_OK +GVL.Pro4_.Monitor.D_Night_Pro_OK[i_qty];
	GVL.Pro4_.Monitor.Total_Day_NG_VS := GVL.Pro4_.Monitor.Total_Day_NG_VS + GVL.Pro4_.Monitor.D_Day_Pro_NG_VS[i_qty];
	GVL.Pro4_.Monitor.Total_Night_NG_VS := GVL.Pro4_.Monitor.Total_Night_NG_VS + GVL.Pro4_.Monitor.D_Night_Pro_NG_VS[i_qty];
	GVL.Pro4_.Monitor.Total_Day_NG_TS := GVL.Pro4_.Monitor.Total_Day_NG_TS + GVL.Pro4_.Monitor.D_Day_Pro_NG_TS[i_qty];
	GVL.Pro4_.Monitor.Total_Night_NG_TS := GVL.Pro4_.Monitor.Total_Night_NG_TS +GVL.Pro4_.Monitor.D_Night_Pro_NG_TS[i_qty];
END_FOR
GVL.Pro4_.Monitor.Total_Day_NG := GVL.Pro4_.Monitor.Total_Day_NG_VS + GVL.Pro4_.Monitor.Total_Day_NG_TS;
GVL.Pro4_.Monitor.Total_Night_NG := GVL.Pro4_.Monitor.Total_Night_NG_VS + GVL.Pro4_.Monitor.Total_Night_NG_TS;
GVL.Pro4_.Monitor.Total_Day := GVL.Pro4_.Monitor.Total_Day_OK + GVL.Pro4_.Monitor.Total_Day_NG;
GVL.Pro4_.Monitor.Total_Night := GVL.Pro4_.Monitor.Total_Night_OK + GVL.Pro4_.Monitor.Total_Night_NG;
GVL.Pro4_.Monitor.All_Shift_OK := GVL.Pro4_.Monitor.Total_Day_OK + GVL.Pro4_.Monitor.Total_Night_OK;
GVL.Pro4_.Monitor.All_Shift_NG := GVL.Pro4_.Monitor.Total_Day_NG + GVL.Pro4_.Monitor.Total_Night_NG;
GVL.Pro4_.Monitor.All_Shift := GVL.Pro4_.Monitor.Total_Day + GVL.Pro4_.Monitor.Total_Night;
END_ACTION

ACTION Tactime_Input:
// Pulse_In := POU_MOTION.Place_B4_Finish;
// T1(IN := POU_MOTION.RUN_PROJECT, PT := T#1H);   // chạy free-run (1h cho khỏi overflow sớm)
// 
// // lấy thời gian đã trôi qua
//     Tact_ms := TO_DWORD(T1.ET)/100;
// IF (Pulse_In = TRUE) AND (Pulse_Old = FALSE) THEN
// 	
// 
// 
//     // reset timer để đo lần tiếp theo
//     T1(IN := FALSE);
//     T1(IN := TRUE);
// 
//     // ===== DỊCH MẢNG =====
//     FOR i_tactime_input := 9 TO 1 BY -1 DO
//         Tact_Array[i_tactime_input] := Tact_Array[i_tactime_input-1];
//     END_FOR
// 
//     // ===== GHI GIÁ TRỊ MỚI NHẤT =====
//     Tact_Array[0] := TO_WORD(Tact_ms);
// 
//     // đếm số mẫu
//     IF Count < 10 THEN
//         Count := Count + 1;
//     END_IF
// 
// END_IF
// 
// Pulse_Old := Pulse_In;

//namnv1104

// Pulse_In := POU_MOTION.Place_B4_Finish;
// Pulse_Out := POU_MOTION.Place_B4_Finish;
T1(PT := T#1H);   // chạy free-run (1h cho khỏi overflow sớm)
IF Pulse_In THEN
	T1.IN := TRUE;
END_IF
// lấy thời gian đã trôi qua
Tact_ms := TO_DWORD(T1.ET)/100;
IF (Pulse_Out = TRUE) AND (Pulse_In = FALSE) AND (Pulse_Old = FALSE) THEN
	
	

    // reset timer để đo lần tiếp theo
    T1(IN := FALSE);
    //T1(IN := TRUE);

    // ===== DỊCH MẢNG =====
    FOR i_tactime_input := 9 TO 1 BY -1 DO
        Tact_Array[i_tactime_input] := Tact_Array[i_tactime_input-1];
    END_FOR

    // ===== GHI GIÁ TRỊ MỚI NHẤT =====
    Tact_Array[0] := TO_WORD(Tact_ms);

    // đếm số mẫu
    IF Count < 10 THEN
        Count := Count + 1;
    END_IF
END_IF

Pulse_Old := Pulse_Out;


/// Avg tactime
Sum_Tact := 0;

FOR i_tactime_input := 0 TO Count - 1 DO
    Sum_Tact := Sum_Tact + Tact_Array[i_tactime_input];
END_FOR

IF Count > 0 THEN
    Avg_Tact := Sum_Tact / Count;
END_IF
END_ACTION

ACTION Tactime_MC1:
// Pulse_In_1 := (POU_MOTION.Pro_MC1_4 = 20) ;
// 
// T2(IN := POU_MOTION.RUN_PROJECT, PT := T#1H);   // chạy free-run (1h cho khỏi overflow sớm)
// 
// // lấy thời gian đã trôi qua
//     Tact_ms_1 := TO_DWORD(T2.ET)/100;
// IF (Pulse_In_1 = TRUE) AND (Pulse_Old_1 = FALSE) THEN
// 	
// 
// 
//     // reset timer để đo lần tiếp theo
//     T2(IN := FALSE);
//     T2(IN := TRUE);
// 
//     // ===== DỊCH MẢNG =====
//     FOR i_tactime_input_1 := 9 TO 1 BY -1 DO
//         Tact_Array_1[i_tactime_input_1] := Tact_Array_1[i_tactime_input_1-1];
//     END_FOR
// 
//     // ===== GHI GIÁ TRỊ MỚI NHẤT =====
//     Tact_Array_1[0] := TO_WORD(Tact_ms_1);
// 
//     // đếm số mẫu
//     IF Count_1 < 10 THEN
//         Count_1 := Count_1 + 1;
//     END_IF
// 
// END_IF
// 
// Pulse_Old_1 := Pulse_In_1;

// Pulse_In_1 := (POU_MOTION.Pro_MC1_4 = 20) ;

T2(PT := T#1H);   // chạy free-run (1h cho khỏi overflow sớm)
IF Pulse_In_1 THEN
	T2.IN := TRUE;
END_IF
// lấy thời gian đã trôi qua
    Tact_ms_1 := TO_DWORD(T2.ET)/100;
IF (Pulse_Out_1 = TRUE) AND (Pulse_Old_1 = FALSE) THEN
	

	
    // reset timer để đo lần tiếp theo
    T2(IN := FALSE);
    //T2(IN := TRUE);

    // ===== DỊCH MẢNG =====
    FOR i_tactime_input_1 := 9 TO 1 BY -1 DO
        Tact_Array_1[i_tactime_input_1] := Tact_Array_1[i_tactime_input_1-1];
    END_FOR

    // ===== GHI GIÁ TRỊ MỚI NHẤT =====
    Tact_Array_1[0] := TO_WORD(Tact_ms_1);

    // đếm số mẫu
    IF Count_1 < 10 THEN
        Count_1 := Count_1 + 1;
    END_IF

END_IF

Pulse_Old_1 := Pulse_Out_1;


/// Avg tactime
Sum_Tact_1 := 0;

FOR i_tactime_input_1 := 0 TO Count_1 - 1 DO
    Sum_Tact_1 := Sum_Tact_1 + Tact_Array_1[i_tactime_input_1];
END_FOR

IF Count_1 > 0 THEN
    Avg_Tact_1 := Sum_Tact_1 / Count_1;
END_IF
END_ACTION

ACTION Tactime_MC2:
// Pulse_In_2 := (POU_MOTION.Pro_MC2_4 = 20) ;
// 
// T3(IN := POU_MOTION.RUN_PROJECT, PT := T#1H);   // chạy free-run (1h cho khỏi overflow sớm)
// 
// // lấy thời gian đã trôi qua
//     Tact_ms_2 := TO_DWORD(T3.ET)/100;
// IF (Pulse_In_2 = TRUE) AND (Pulse_Old_2 = FALSE) THEN
// 	
// 
// 
//     // reset timer để đo lần tiếp theo
//     T3(IN := FALSE);
//     T3(IN := TRUE);
// 
//     // ===== DỊCH MẢNG =====
//     FOR i_tactime_input_2 := 9 TO 1 BY -1 DO
//         Tact_Array_2[i_tactime_input_2] := Tact_Array_2[i_tactime_input_2-1];
//     END_FOR
// 
//     // ===== GHI GIÁ TRỊ MỚI NHẤT =====
//     Tact_Array_2[0] := TO_WORD(Tact_ms_2) ;
// 
//     // đếm số mẫu
//     IF Count_2 < 10 THEN
//         Count_2 := Count_2 + 1;
//     END_IF
// 
// END_IF
// 
// Pulse_Old_2 := Pulse_In_2;

// Pulse_In_2 := (POU_MOTION.Pro_MC2_4 = 20) ;

T3(PT := T#1H);   // chạy free-run (1h cho khỏi overflow sớm)
IF Pulse_In_2 THEN
	T3.IN := TRUE;
END_IF
// lấy thời gian đã trôi qua
    Tact_ms_2 := TO_DWORD(T3.ET)/100;
IF (Pulse_Out_2 = TRUE) AND (Pulse_Old_2 = FALSE) THEN
	
	
    // reset timer để đo lần tiếp theo
    T3(IN := FALSE);
    //T3(IN := TRUE);

    // ===== DỊCH MẢNG =====
    FOR i_tactime_input_2 := 9 TO 1 BY -1 DO
        Tact_Array_2[i_tactime_input_2] := Tact_Array_2[i_tactime_input_2-1];
    END_FOR

    // ===== GHI GIÁ TRỊ MỚI NHẤT =====
    Tact_Array_2[0] := TO_WORD(Tact_ms_2) ;

    // đếm số mẫu
    IF Count_2 < 10 THEN
        Count_2 := Count_2 + 1;
    END_IF

END_IF

Pulse_Old_2 := Pulse_Out_2;


/// Avg tactime
Sum_Tact_2 := 0;

FOR i_tactime_input_2 := 0 TO Count_2 - 1 DO
    Sum_Tact_2 := Sum_Tact_2 + Tact_Array_2[i_tactime_input_2];
END_FOR

IF Count_2 > 0 THEN
    Avg_Tact_2 := Sum_Tact_2 / Count_2;
END_IF
END_ACTION

ACTION Tactime_output:
// Pulse_In_ := (POU_MOTION.Place_NG_A4_T2_Finish OR POU_MOTION.Place_NG_TS_A4_T2_Finish OR  POU_MOTION.Place_NG_A4_T2_Finish) ; ;
// T4(IN := POU_MOTION.RUN_PROJECT, PT := T#1H);   // chạy free-run (1h cho khỏi overflow sớm)
// 
// // lấy thời gian đã trôi qua
//     Tact_ms_ := TO_DWORD(T4.ET)/100;
// IF (Pulse_In_ = TRUE) AND (Pulse_Old_ = FALSE) THEN
// 	
// 
// 
//     // reset timer để đo lần tiếp theo
//     T4(IN := FALSE);
//     T4(IN := TRUE);
// 
//     // ===== DỊCH MẢNG =====
//     FOR i_tactime_input_ := 9 TO 1 BY -1 DO
//         Tact_Array_[i_tactime_input_] := Tact_Array_[i_tactime_input_-1];
//     END_FOR
// 
//     // ===== GHI GIÁ TRỊ MỚI NHẤT =====
//     Tact_Array_[0] := TO_WORD(Tact_ms_);
// 
//     // đếm số mẫu
//     IF Count_ < 10 THEN
//         Count_ := Count_ + 1;
//     END_IF
// 
// END_IF
// 
// Pulse_Old_ := Pulse_In_;

// Pulse_In_ := (POU_MOTION.Place_NG_A4_T2_Finish OR POU_MOTION.Place_NG_TS_A4_T2_Finish OR  POU_MOTION.Place_NG_A4_T2_Finish);

T4(PT := T#1H);   // chạy free-run (1h cho khỏi overflow sớm)

IF Pulse_In_ THEN
	T4.IN := TRUE;
END_IF
// lấy thời gian đã trôi qua
Tact_ms_ := TO_DWORD(T4.ET)/100;
IF (Pulse_Out_ = TRUE) AND (Pulse_In_ = FALSE) AND (Pulse_Old_ = FALSE) THEN
	
	

    // reset timer để đo lần tiếp theo
    T4(IN := FALSE);
    //T4(IN := TRUE);

    // ===== DỊCH MẢNG =====
    FOR i_tactime_input_ := 9 TO 1 BY -1 DO
        Tact_Array_[i_tactime_input_] := Tact_Array_[i_tactime_input_ - 1];
    END_FOR

    // ===== GHI GIÁ TRỊ MỚI NHẤT =====
    Tact_Array_[0] := TO_WORD(Tact_ms_);

    // đếm số mẫu
    IF Count_ < 10 THEN
        Count_ := Count_ + 1;
    END_IF

END_IF

Pulse_Old_ := Pulse_Out_;


/// Avg tactime
Sum_Tact_ := 0;

FOR i_tactime_input_ := 0 TO Count_ - 1 DO
    Sum_Tact_ := Sum_Tact_ + Tact_Array_[i_tactime_input_];
END_FOR

IF Count_ > 0 THEN
    Avg_Tact_ := Sum_Tact_ / Count_;
END_IF
END_ACTION

END_PROGRAM

// Just_Motion_Control_x86_64_Linux_SM_WV/Application/PRG_ROBOT/POU_HMI_CONTROL_ROBOT
PROGRAM POU_HMI_CONTROL_ROBOT
VAR
	SR1,SR2,SR3,SR4,SR5,SR6,SR7,SR8,
	SR_HMI_CONTROL_PANEL_1, SR_JOG_AND_TEACH_1,SR_POINT_1,SR_TOOLS_1,SR_PALLETS_1,SR_XYZ_LIMIT_1, SR_ROBOT_CONFIG_1,
	SR_HMI_CONTROL_PANEL_2, SR_JOG_AND_TEACH_2,SR_POINT_2,SR_TOOLS_2,SR_PALLETS_2,SR_XYZ_LIMIT_2, SR_ROBOT_CONFIG_2 : SR;
	RS_JOG_CONTINUE_1, RS_JOG_INCHING_1, RS_JOG_POINT_1,
	RS_JOG_CONTINUE_2, RS_JOG_INCHING_2, RS_JOG_POINT_2 : SR;
	TRIG_JOG_CONTINUE_1, TRIG_JOG_INCHING_1, TRIG_JOG_POINT_1,
	TRIG_JOG_CONTINUE_2, TRIG_JOG_INCHING_2, TRIG_JOG_POINT_2 : R_TRIG;
	
	D_HMI_SCREEN , D_PLC_SCREEN : WORD;
	D_SELECT_RB, D_SELECT_TOOL_RB_A, D_SELECT_TOOL_RB_B : WORD;

	R_TRIG_0, R_TRIG_1, R_TRIG_2: R_TRIG;

	PrevSelectRB : WORD;
END_VAR

VAR // act_manORauto
	TR_MAN, TR_AUTO , TR_MAN_AB, TR_AUTO_AB : R_TRIG;
	
END_VAR
VAR
	i, idx, iPoint : INT;
END_VAR

// HMI Edit Point
VAR
	Delete_all_point, Delete_one_point : TON;
	Delete_all_Step, Delete_one_Step : TON;
END_VAR

// HMI Condition
VAR
    condNo : INT;
    rowNo : INT;
	rowResult : BOOL;
    finalResult : BOOL;
    firstRow : BOOL;
END_VAR

// ============================================================
// ADD LOCAL VARIABLES TO POU_HMI_CONTROL_ROBOT
// Không dùng chung TON A/B vì hai editor có thể được scan cùng lúc.
// ============================================================
VAR
    Delete_all_point_B : TON;
    Delete_one_point_B : TON;
    Delete_all_Step_B : TON;
    Delete_one_Step_B : TON;
END_VAR
VAR // added by the converter: edge detectors and wires of the graphical bodies
    _w1 : BOOL;
END_VAR

// DEFINT
ACT_View_Edit_Point_A();
ACT_View_Edit_Cmd();
ACT_HMI_A_ConditionEditor();
ACT_HMIToolConfigEditor_A();
ACT_HMI_SensorSource_Config();
ACT_HMI_Recipe_Config();
ACT_HMI_A_Vision_Tracking_Config();

// ============================================================
ACT_View_Edit_Point_B();
ACT_View_Edit_Cmd_B();
ACT_HMI_B_ConditionEditor();

ACT_HMIToolConfigEditor_B();
ACT_HMI_SensorSource_Config_B();
ACT_HMI_Recipe_Config_B();
ACT_HMI_B_Vision_Tracking_Config();


ACT_select_rb();
ACT_MANORAUTO();
ACT_MENU();
ACT_ControlPanel();
ACT_JOG_LOGIC();
// Read Window
D_HMI_SCREEN := GVL.DW_[2]; // O NHO CHUA SO PAGE CỦA HMI
GVL.DW_[4] := D_PLC_SCREEN; // THAY ĐỔI TRANG HMI TỪ PLC
D_SELECT_RB := GVL.DW_[0]; // SELECT ROBOT TRONG H
/// RESET DATA 1
SR_HMI_CONTROL_PANEL_1(SET1 := D_HMI_SCREEN = 20,
	RESET := D_HMI_SCREEN <> 20,
	Q1 => GVL.MB_[20]);
SR_JOG_AND_TEACH_1(SET1 := D_HMI_SCREEN = 21,
	RESET := D_HMI_SCREEN <> 21,
	Q1 => GVL.MB_[21]);
SR_POINT_1(SET1 := D_HMI_SCREEN = 22 OR D_HMI_SCREEN = 120 OR D_HMI_SCREEN = 121 OR D_HMI_SCREEN = 122 OR D_HMI_SCREEN = 123,
	RESET := D_HMI_SCREEN <> 22 AND D_HMI_SCREEN <> 120 AND D_HMI_SCREEN <> 121 AND D_HMI_SCREEN <> 122 AND D_HMI_SCREEN <> 123,
	Q1 => GVL.MB_[22]);
SR_TOOLS_1(SET1 := D_HMI_SCREEN = 23,
	RESET := D_HMI_SCREEN <> 23,
	Q1 => GVL.MB_[23]);
SR_PALLETS_1(SET1 := D_HMI_SCREEN = 24,
	RESET := D_HMI_SCREEN <> 24,
	Q1 => GVL.MB_[24]);
SR_XYZ_LIMIT_1(SET1 := D_HMI_SCREEN = 25 OR D_HMI_SCREEN = 110,
	RESET := D_HMI_SCREEN <> 25 AND D_HMI_SCREEN <> 110,
	Q1 => GVL.MB_[25]);	
SR_ROBOT_CONFIG_1(SET1 := D_HMI_SCREEN = 26,
	RESET := D_HMI_SCREEN <> 26,
	Q1 => GVL.MB_[26]);			
/// RESET DATA 2
SR_HMI_CONTROL_PANEL_2(SET1 := D_HMI_SCREEN = 30,
	RESET := D_HMI_SCREEN <> 30,
	Q1 => GVL.MB_[30]);
SR_JOG_AND_TEACH_2(SET1 := D_HMI_SCREEN = 31,
	RESET := D_HMI_SCREEN <> 31,
	Q1 => GVL.MB_[31]);
SR_POINT_2(SET1 := D_HMI_SCREEN = 32 OR D_HMI_SCREEN = 130 OR D_HMI_SCREEN = 131 OR D_HMI_SCREEN = 132 OR D_HMI_SCREEN = 133,
	RESET := D_HMI_SCREEN <> 32 AND D_HMI_SCREEN <> 130 AND D_HMI_SCREEN <> 131 AND D_HMI_SCREEN <> 132 AND D_HMI_SCREEN <> 133,
	Q1 => GVL.MB_[32]);
SR_TOOLS_2(SET1 := D_HMI_SCREEN = 33,
	RESET := D_HMI_SCREEN <> 33,
	Q1 => GVL.MB_[33]);
SR_PALLETS_2(SET1 := D_HMI_SCREEN = 34,
	RESET := D_HMI_SCREEN <> 34,
	Q1 => GVL.MB_[34]);
SR_XYZ_LIMIT_2(SET1 := D_HMI_SCREEN = 35 OR D_HMI_SCREEN = 111 ,
	RESET := D_HMI_SCREEN <> 35 AND D_HMI_SCREEN <> 111,
	Q1 => GVL.MB_[35]);	
SR_ROBOT_CONFIG_2(SET1 := D_HMI_SCREEN = 36,
	RESET := D_HMI_SCREEN <> 36,
	Q1 => GVL.MB_[36]);

ACTION ACT_ControlPanel:
/// Control panel 1
SR1(SET1 := gvl.RB_A.Home_Lock_All OR (NOT GVL.RB_A.Home_Free_All AND GVL.RB_A.M1_goHome ) AND D_HMI_SCREEN = 20, 
	RESET:= GVL.RB_A.Home_Free_All OR NOT GVL.RB_A.M1_goHome OR D_HMI_SCREEN <> 20,
	Q1 => GVL.RB_A.M1_goHome);
SR2(SET1 := gvl.RB_A.Home_Lock_All OR (NOT GVL.RB_A.Home_Free_All AND GVL.RB_A.M2_goHome) AND D_HMI_SCREEN = 20, 
	RESET:= GVL.RB_A.Home_Free_All OR NOT GVL.RB_A.M2_goHome OR D_HMI_SCREEN <> 20,
	Q1 => GVL.RB_A.M2_goHome);
SR3(SET1 := gvl.RB_A.Home_Lock_All OR (NOT GVL.RB_A.Home_Free_All AND GVL.RB_A.M3_goHome) AND D_HMI_SCREEN = 20, 
	RESET:= GVL.RB_A.Home_Free_All OR NOT GVL.RB_A.M3_goHome OR D_HMI_SCREEN <> 20,
	Q1 => GVL.RB_A.M3_goHome);
SR4(SET1 := gvl.RB_A.Home_Lock_All OR (NOT GVL.RB_A.Home_Free_All AND GVL.RB_A.M4_goHome) AND D_HMI_SCREEN = 20, 
	RESET:= GVL.RB_A.Home_Free_All OR NOT GVL.RB_A.M4_goHome OR D_HMI_SCREEN <> 20,
	Q1 => GVL.RB_A.M4_goHome);
/// Control panel 2
SR5(SET1 := gvl.RB_B.Home_Lock_All OR (NOT GVL.RB_B.Home_Free_All AND GVL.RB_B.M1_goHome) AND D_HMI_SCREEN = 30, 
	RESET:= GVL.RB_B.Home_Free_All OR NOT GVL.RB_B.M1_goHome OR D_HMI_SCREEN <> 30,
	Q1 => GVL.RB_B.M1_goHome);
SR6(SET1 := gvl.RB_B.Home_Lock_All OR (NOT GVL.RB_B.Home_Free_All AND GVL.RB_B.M2_goHome) AND D_HMI_SCREEN = 30, 
	RESET:= GVL.RB_B.Home_Free_All OR NOT GVL.RB_B.M2_goHome OR D_HMI_SCREEN <> 30,
	Q1 => GVL.RB_B.M2_goHome);
SR7(SET1 := gvl.RB_B.Home_Lock_All OR (NOT GVL.RB_B.Home_Free_All AND GVL.RB_B.M3_goHome) AND D_HMI_SCREEN = 30, 
	RESET:= GVL.RB_B.Home_Free_All OR NOT GVL.RB_B.M3_goHome OR D_HMI_SCREEN <> 30,
	Q1 => GVL.RB_B.M3_goHome);
SR8(SET1 := gvl.RB_B.Home_Lock_All OR (NOT GVL.RB_B.Home_Free_All AND GVL.RB_B.M4_goHome) AND D_HMI_SCREEN = 30, 
	RESET:= GVL.RB_B.Home_Free_All OR NOT GVL.RB_B.M4_goHome OR D_HMI_SCREEN <> 30,
	Q1 => GVL.RB_B.M4_goHome);
END_ACTION

ACTION ACT_HMI_A_ConditionEditor:
//====================================================
// PRG_HMI_A_ConditionEditor
// Hiển thị danh sách condition + xử lý Load/Save/Edit
//====================================================

// Scroll danh sách condition
IF GVL.HMI_A_CondCmd_Up THEN
    GVL.HMI_A_CondCmd_Up := FALSE;
    IF GVL.HMI_A_CondViewStart > 1 THEN
        GVL.HMI_A_CondViewStart := GVL.HMI_A_CondViewStart - 1;
    END_IF;
END_IF;

IF GVL.HMI_A_CondCmd_Down THEN
    GVL.HMI_A_CondCmd_Down := FALSE;
    IF GVL.HMI_A_CondViewStart < 91 THEN
        GVL.HMI_A_CondViewStart := GVL.HMI_A_CondViewStart + 1;
    END_IF;
END_IF;

IF GVL.HMI_A_CondCmd_PageUp THEN
    GVL.HMI_A_CondCmd_PageUp := FALSE;
    GVL.HMI_A_CondViewStart := GVL.HMI_A_CondViewStart - 10;
    IF GVL.HMI_A_CondViewStart < 1 THEN
        GVL.HMI_A_CondViewStart := 1;
    END_IF;
END_IF;

IF GVL.HMI_A_CondCmd_PageDown THEN
    GVL.HMI_A_CondCmd_PageDown := FALSE;
    GVL.HMI_A_CondViewStart := GVL.HMI_A_CondViewStart + 10;
    IF GVL.HMI_A_CondViewStart > 91 THEN
        GVL.HMI_A_CondViewStart := 91;
    END_IF;
END_IF;

IF GVL.HMI_A_CondCmd_GoTop THEN
    GVL.HMI_A_CondCmd_GoTop := FALSE;
    GVL.HMI_A_CondViewStart := 1;
END_IF;

IF GVL.HMI_A_CondCmd_GoBot THEN
    GVL.HMI_A_CondCmd_GoBot := FALSE;
    GVL.HMI_A_CondViewStart := 91;
END_IF;


//====================================================
// Row Select
//====================================================

FOR i := 1 TO 10 DO
    IF (GVL.HMI_A_CondSelectedCmd = i) THEN
		GVL.HMI_A_CondRowSelect[i] := TRUE;
		GVL.HMI_A_CondSelectedNo := i + GVL.HMI_A_CondViewStart - 1;
		//GVL.HMI_A_EditStepNo   := GVL.HMI_A_SelectedStepNo;
	ELSE
		GVL.HMI_A_CondRowSelect[i] := FALSE;
    END_IF;
END_FOR;

// FOR i := 1 TO 10 DO
//     IF GVL.HMI_A_CondRowSelect[i] THEN
//         GVL.HMI_A_CondRowSelect[i] := FALSE;
//         condNo := GVL.HMI_A_CondViewNo[i];
// 
//         IF (condNo >= 1) AND (condNo <= 100) THEN
//             GVL.HMI_A_CondSelectedNo := condNo;
//             GVL.HMI_A_CondCmdReq := 1; // Load
//         END_IF;
//     END_IF;
// END_FOR;


//====================================================
// Update View 10 dòng condition
//====================================================
FOR i := 1 TO 10 DO
    condNo := GVL.HMI_A_CondViewStart + i - 1;

    IF (condNo >= 1) AND (condNo <= 100) THEN
        GVL.HMI_A_CondViewNo[i]     := condNo;
        GVL.HMI_A_CondViewName[i]   := GVL_1.Condition_Cr_A[condNo].Name;
        GVL.HMI_A_CondViewEnable[i] := GVL_1.Condition_Cr_A[condNo].Enable;
        GVL.HMI_A_CondViewResult[i] := GVL_1.Condition_Cr_A[condNo].Result;
    ELSE
        GVL.HMI_A_CondViewNo[i]     := 0;
        GVL.HMI_A_CondViewName[i]   := '';
        GVL.HMI_A_CondViewEnable[i] := FALSE;
        GVL.HMI_A_CondViewResult[i] := FALSE;
    END_IF;
END_FOR;


//====================================================
// Command Load / Save / Clear / Copy / Paste
//====================================================
CASE GVL.HMI_A_CondCmdReq OF

    1: // Load condition vào vùng Edit
        condNo := GVL.HMI_A_CondSelectedNo;

        IF (condNo >= 1) AND (condNo <= 100) THEN
            GVL.HMI_A_CondEditNo := condNo;
            GVL.HMI_A_CondEditName := GVL_1.Condition_Cr_A[condNo].Name;
            GVL.HMI_A_CondEditEnable := GVL_1.Condition_Cr_A[condNo].Enable;

            FOR i := 1 TO 10 DO
                GVL.HMI_A_CondEditRowEnable[i] := GVL_1.Condition_Cr_A[condNo].Row[i].Enable;
                GVL.HMI_A_CondEditSource[i]    := GVL_1.Condition_Cr_A[condNo].Row[i].Source;
                GVL.HMI_A_CondEditIndex[i]     := GVL_1.Condition_Cr_A[condNo].Row[i].Index;
                GVL.HMI_A_CondEditOperator[i]  := GVL_1.Condition_Cr_A[condNo].Row[i].Operator;
                GVL.HMI_A_CondEditSetValue[i]  := GVL_1.Condition_Cr_A[condNo].Row[i].SetValue;
                GVL.HMI_A_CondEditLinkNext[i]  := GVL_1.Condition_Cr_A[condNo].Row[i].LinkNext;
                //GVL.HMI_A_CondEditNote[i]      := GVL_1.Condition_Cr_A[condNo].Row[i].Note;
            END_FOR;
        END_IF;

        GVL.HMI_A_CondCmdReq := 0;


    2: // Save vùng Edit về bảng thật
        condNo := GVL.HMI_A_CondSelectedNo;

        IF (condNo >= 1) AND (condNo <= 100) THEN
            GVL_1.Condition_Cr_A[condNo].Name := GVL.HMI_A_CondEditName;
            GVL_1.Condition_Cr_A[condNo].Enable := GVL.HMI_A_CondEditEnable;

